// TIA Portal V15.1 export
// export: Created 2024-06-21T08:41:24.854849Z, ExportSetting WithDefaults, DisplayName Totally Integrated Automation Portal, DisplayVersion V15.1 Update 5, DisplayName TIA Portal Openness, DisplayVersion V15.1 Update 5, DisplayName SINAMICS Startdrive Advanced, DisplayVersion V15.1, DisplayName G130, G150, S120, S150, SINAMICS MV, S210, DisplayVersion V15.1, DisplayName G110M, G120, G120C, G120D, G120P, DisplayVersion V15.1, DisplayName STEP 7 Professional, DisplayVersion V15.1 Update 5, DisplayName STEP 7 Safety, DisplayVersion V15.1, DisplayName WinCC Professional, DisplayVersion V15.1 Update 5, DisplayName SIMATIC Visualization Architect, DisplayVersion V15.1
FUNCTION "209230ZM01" : Void   // FC400, FBD
TITLE = 209230ZM01 ModeZone
{ S7_Optimized_Access := 'FALSE' }
AUTHOR : VCG
NAME : Mot001
VERSION : 0.1
// stored: AutoNumber false, IsIECCheckEnabled false, SetENOAutomatically False, UDAEnableTagReadback false
   VAR_OUTPUT
      O_AlarmA : Bool;   // Alarm A
      O_AlarmB : Bool;   // Alarm B
      O_AlarmC : Bool;   // Alarm C
      O_AlarmD : Bool;   // Alarm D
      O_AlarmABCondition : Bool;   // Alarms resetable
      H_IAnim : Word;   // Animation bits to Icon in WinCC
   END_VAR
   VAR_TEMP   // added for the SCL form of the ladder/FBD networks
      _w1 : Bool;
      _w2 : Bool;
   END_VAR
BEGIN

REGION Network 1: **** 1 - Inputs **** HMI Commands
   // HMI Commands from the WinCC
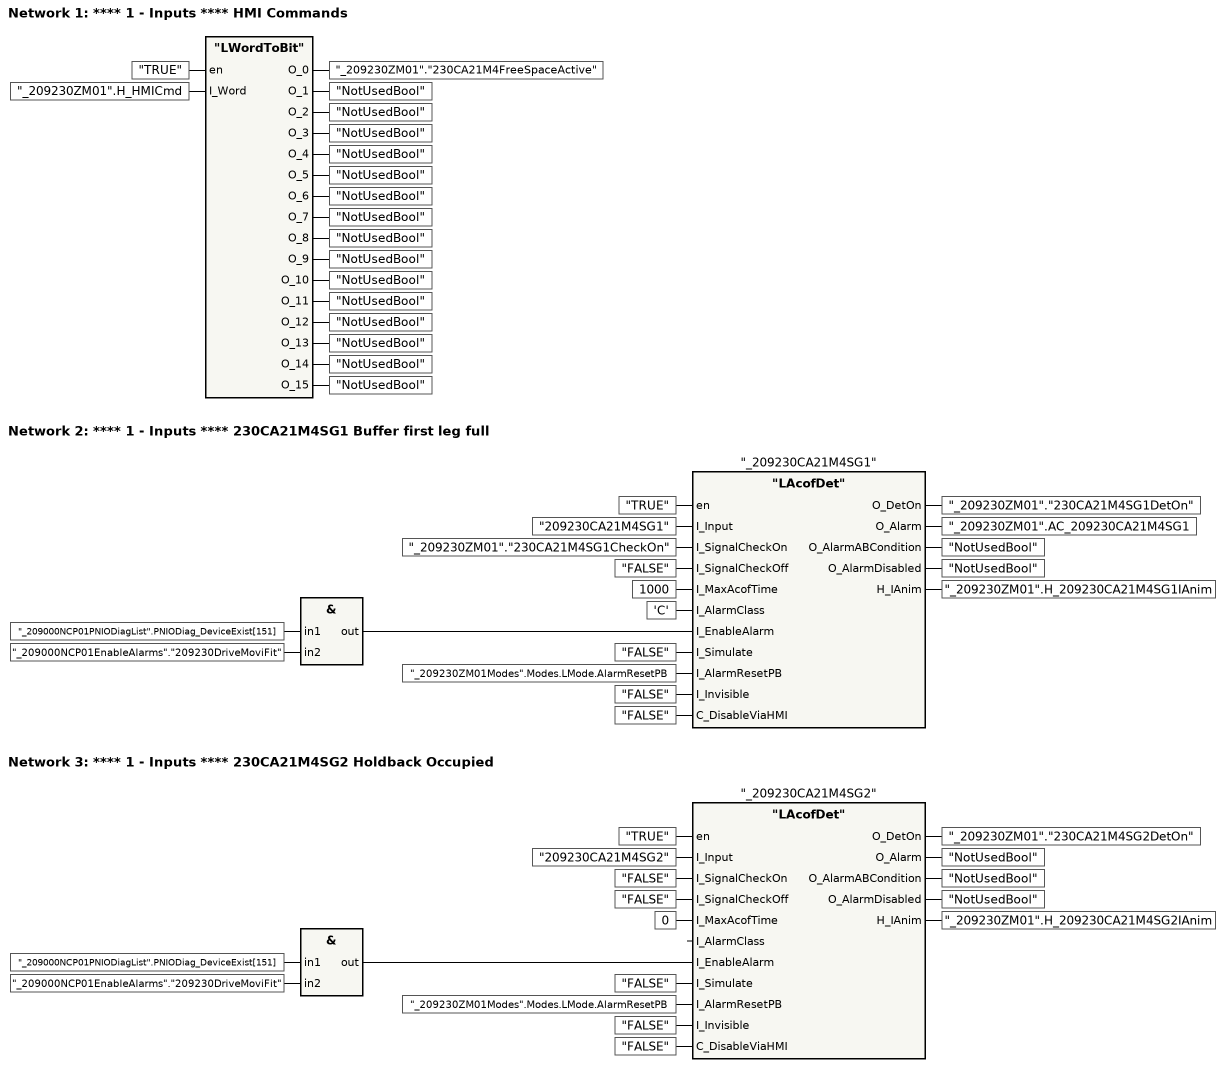
   IF "TRUE" THEN
       "LWordToBit"(I_Word := "_209230ZM01".H_HMICmd,
                    O_0 => "_209230ZM01"."230CA21M4FreeSpaceActive",
                    O_1 => "NotUsedBool",
                    O_2 => "NotUsedBool",
                    O_3 => "NotUsedBool",
                    O_4 => "NotUsedBool",
                    O_5 => "NotUsedBool",
                    O_6 => "NotUsedBool",
                    O_7 => "NotUsedBool",
                    O_8 => "NotUsedBool",
                    O_9 => "NotUsedBool",
                    O_10 => "NotUsedBool",
                    O_11 => "NotUsedBool",
                    O_12 => "NotUsedBool",
                    O_13 => "NotUsedBool",
                    O_14 => "NotUsedBool",
                    O_15 => "NotUsedBool");
   END_IF;
END_REGION

REGION Network 2: **** 1 - Inputs **** 230CA21M4SG1 Buffer first leg full
   IF "TRUE" THEN
       "_209230CA21M4SG1"(I_Input := "209230CA21M4SG1",   // "LAcofDet"
                          I_SignalCheckOn := "_209230ZM01"."230CA21M4SG1CheckOn",
                          I_SignalCheckOff := "FALSE",
                          I_MaxAcofTime := 1000,
                          I_AlarmClass := 'C',
                          I_EnableAlarm := "_209000NCP01PNIODiagList".PNIODiag_DeviceExist[151] AND "_209000NCP01EnableAlarms"."209230DriveMoviFit",
                          I_Simulate := "FALSE",
                          I_AlarmResetPB := "_209230ZM01Modes".Modes.LMode.AlarmResetPB,
                          I_Invisible := "FALSE",
                          C_DisableViaHMI := "FALSE",
                          O_DetOn => "_209230ZM01"."230CA21M4SG1DetOn",
                          O_Alarm => "_209230ZM01".AC_209230CA21M4SG1,
                          O_AlarmABCondition => "NotUsedBool",
                          O_AlarmDisabled => "NotUsedBool",
                          H_IAnim => "_209230ZM01".H_209230CA21M4SG1IAnim);
   END_IF;
END_REGION

REGION Network 3: **** 1 - Inputs **** 230CA21M4SG2 Holdback Occupied
   IF "TRUE" THEN
       "_209230CA21M4SG2"(I_Input := "209230CA21M4SG2",   // "LAcofDet"
                          I_SignalCheckOn := "FALSE",
                          I_SignalCheckOff := "FALSE",
                          I_MaxAcofTime := 0,
                          I_EnableAlarm := "_209000NCP01PNIODiagList".PNIODiag_DeviceExist[151] AND "_209000NCP01EnableAlarms"."209230DriveMoviFit",
                          I_Simulate := "FALSE",
                          I_AlarmResetPB := "_209230ZM01Modes".Modes.LMode.AlarmResetPB,
                          I_Invisible := "FALSE",
                          C_DisableViaHMI := "FALSE",
                          O_DetOn => "_209230ZM01"."230CA21M4SG2DetOn",
                          O_Alarm => "NotUsedBool",
                          O_AlarmABCondition => "NotUsedBool",
                          O_AlarmDisabled => "NotUsedBool",
                          H_IAnim => "_209230ZM01".H_209230CA21M4SG2IAnim);
   END_IF;
END_REGION

REGION Network 4: **** 1 - Inputs **** 230CA21M4SG3 OK to close Holdback
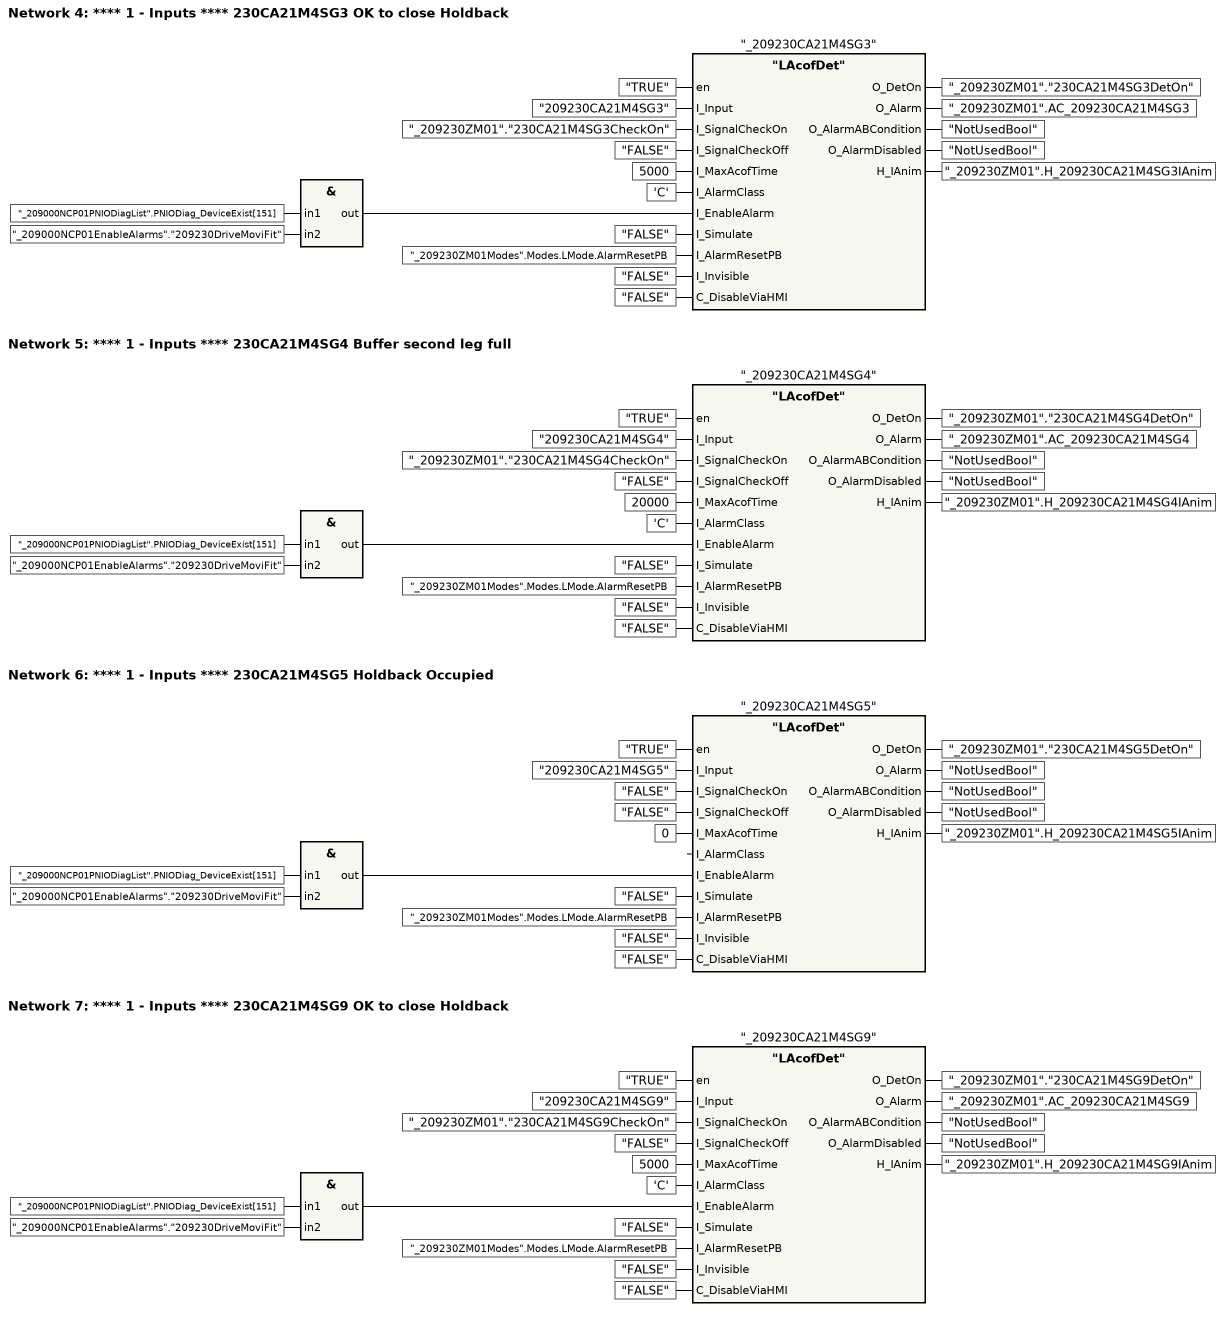
   IF "TRUE" THEN
       "_209230CA21M4SG3"(I_Input := "209230CA21M4SG3",   // "LAcofDet"
                          I_SignalCheckOn := "_209230ZM01"."230CA21M4SG3CheckOn",
                          I_SignalCheckOff := "FALSE",
                          I_MaxAcofTime := 5000,
                          I_AlarmClass := 'C',
                          I_EnableAlarm := "_209000NCP01PNIODiagList".PNIODiag_DeviceExist[151] AND "_209000NCP01EnableAlarms"."209230DriveMoviFit",
                          I_Simulate := "FALSE",
                          I_AlarmResetPB := "_209230ZM01Modes".Modes.LMode.AlarmResetPB,
                          I_Invisible := "FALSE",
                          C_DisableViaHMI := "FALSE",
                          O_DetOn => "_209230ZM01"."230CA21M4SG3DetOn",
                          O_Alarm => "_209230ZM01".AC_209230CA21M4SG3,
                          O_AlarmABCondition => "NotUsedBool",
                          O_AlarmDisabled => "NotUsedBool",
                          H_IAnim => "_209230ZM01".H_209230CA21M4SG3IAnim);
   END_IF;
END_REGION

REGION Network 5: **** 1 - Inputs **** 230CA21M4SG4 Buffer second leg full
   IF "TRUE" THEN
       "_209230CA21M4SG4"(I_Input := "209230CA21M4SG4",   // "LAcofDet"
                          I_SignalCheckOn := "_209230ZM01"."230CA21M4SG4CheckOn",
                          I_SignalCheckOff := "FALSE",
                          I_MaxAcofTime := 20000,
                          I_AlarmClass := 'C',
                          I_EnableAlarm := "_209000NCP01PNIODiagList".PNIODiag_DeviceExist[151] AND "_209000NCP01EnableAlarms"."209230DriveMoviFit",
                          I_Simulate := "FALSE",
                          I_AlarmResetPB := "_209230ZM01Modes".Modes.LMode.AlarmResetPB,
                          I_Invisible := "FALSE",
                          C_DisableViaHMI := "FALSE",
                          O_DetOn => "_209230ZM01"."230CA21M4SG4DetOn",
                          O_Alarm => "_209230ZM01".AC_209230CA21M4SG4,
                          O_AlarmABCondition => "NotUsedBool",
                          O_AlarmDisabled => "NotUsedBool",
                          H_IAnim => "_209230ZM01".H_209230CA21M4SG4IAnim);
   END_IF;
END_REGION

REGION Network 6: **** 1 - Inputs **** 230CA21M4SG5 Holdback Occupied
   IF "TRUE" THEN
       "_209230CA21M4SG5"(I_Input := "209230CA21M4SG5",   // "LAcofDet"
                          I_SignalCheckOn := "FALSE",
                          I_SignalCheckOff := "FALSE",
                          I_MaxAcofTime := 0,
                          I_EnableAlarm := "_209000NCP01PNIODiagList".PNIODiag_DeviceExist[151] AND "_209000NCP01EnableAlarms"."209230DriveMoviFit",
                          I_Simulate := "FALSE",
                          I_AlarmResetPB := "_209230ZM01Modes".Modes.LMode.AlarmResetPB,
                          I_Invisible := "FALSE",
                          C_DisableViaHMI := "FALSE",
                          O_DetOn => "_209230ZM01"."230CA21M4SG5DetOn",
                          O_Alarm => "NotUsedBool",
                          O_AlarmABCondition => "NotUsedBool",
                          O_AlarmDisabled => "NotUsedBool",
                          H_IAnim => "_209230ZM01".H_209230CA21M4SG5IAnim);
   END_IF;
END_REGION

REGION Network 7: **** 1 - Inputs **** 230CA21M4SG9 OK to close Holdback
   IF "TRUE" THEN
       "_209230CA21M4SG9"(I_Input := "209230CA21M4SG9",   // "LAcofDet"
                          I_SignalCheckOn := "_209230ZM01"."230CA21M4SG9CheckOn",
                          I_SignalCheckOff := "FALSE",
                          I_MaxAcofTime := 5000,
                          I_AlarmClass := 'C',
                          I_EnableAlarm := "_209000NCP01PNIODiagList".PNIODiag_DeviceExist[151] AND "_209000NCP01EnableAlarms"."209230DriveMoviFit",
                          I_Simulate := "FALSE",
                          I_AlarmResetPB := "_209230ZM01Modes".Modes.LMode.AlarmResetPB,
                          I_Invisible := "FALSE",
                          C_DisableViaHMI := "FALSE",
                          O_DetOn => "_209230ZM01"."230CA21M4SG9DetOn",
                          O_Alarm => "_209230ZM01".AC_209230CA21M4SG9,
                          O_AlarmABCondition => "NotUsedBool",
                          O_AlarmDisabled => "NotUsedBool",
                          H_IAnim => "_209230ZM01".H_209230CA21M4SG9IAnim);
   END_IF;
END_REGION

REGION Network 8: **** 1 - Inputs **** 230CA21M4 Buffer Full
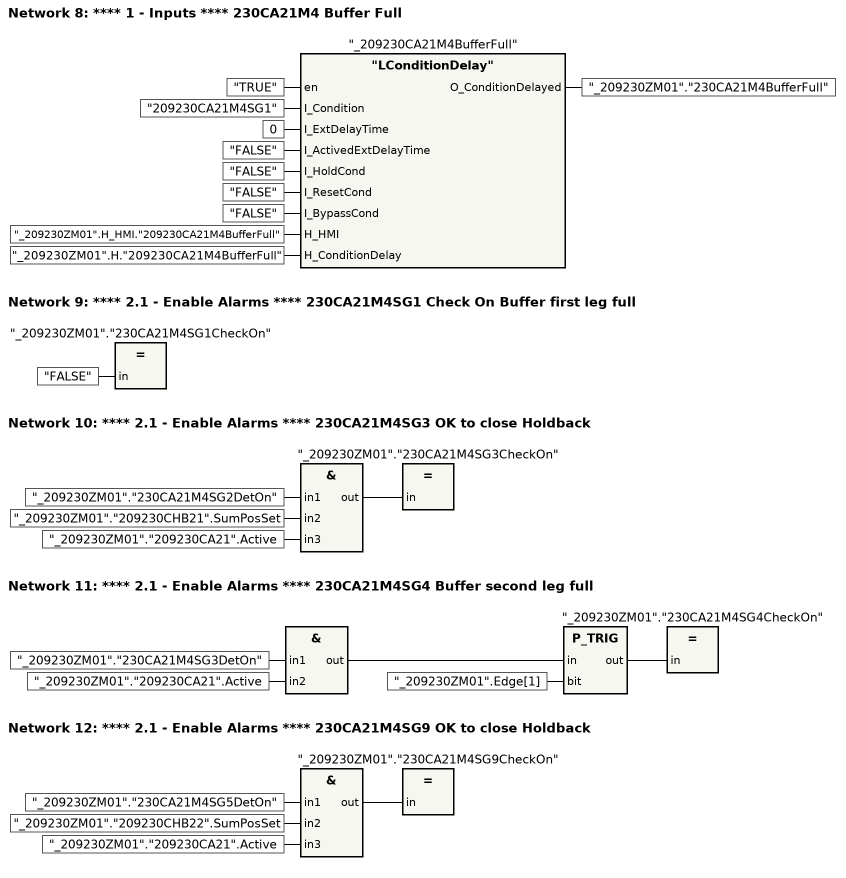
   IF "TRUE" THEN
       "_209230CA21M4BufferFull"(I_Condition := "209230CA21M4SG1",   // "LConditionDelay"
                               I_ExtDelayTime := 0,
                               I_ActivedExtDelayTime := "FALSE",
                               I_HoldCond := "FALSE",
                               I_ResetCond := "FALSE",
                               I_BypassCond := "FALSE",
                               H_HMI := "_209230ZM01".H_HMI."209230CA21M4BufferFull",
                               H_ConditionDelay := "_209230ZM01".H."209230CA21M4BufferFull",
                               O_ConditionDelayed => "_209230ZM01"."230CA21M4BufferFull");
   END_IF;
END_REGION

REGION Network 9: **** 2.1 - Enable Alarms **** 230CA21M4SG1 Check On Buffer first leg full
   "_209230ZM01"."230CA21M4SG1CheckOn" := "FALSE";
END_REGION

REGION Network 10: **** 2.1 - Enable Alarms **** 230CA21M4SG3 OK to close Holdback
   "_209230ZM01"."230CA21M4SG3CheckOn" := "_209230ZM01"."230CA21M4SG2DetOn" AND "_209230ZM01"."209230CHB21".SumPosSet AND "_209230ZM01"."209230CA21".Active;
END_REGION

REGION Network 11: **** 2.1 - Enable Alarms **** 230CA21M4SG4 Buffer second leg full
   #_w1 := "_209230ZM01"."230CA21M4SG3DetOn" AND "_209230ZM01"."209230CA21".Active;
   #_w2 := #_w1 AND NOT "_209230ZM01".Edge[1];   // rising edge
   "_209230ZM01".Edge[1] := #_w1;
   "_209230ZM01"."230CA21M4SG4CheckOn" := #_w2;
END_REGION

REGION Network 12: **** 2.1 - Enable Alarms **** 230CA21M4SG9 OK to close Holdback
   "_209230ZM01"."230CA21M4SG9CheckOn" := "_209230ZM01"."230CA21M4SG5DetOn" AND "_209230ZM01"."209230CHB22".SumPosSet AND "_209230ZM01"."209230CA21".Active;
END_REGION

REGION Network 13: **** 3.1 - Communication - Other Systems **** Supervision
   // Supervision
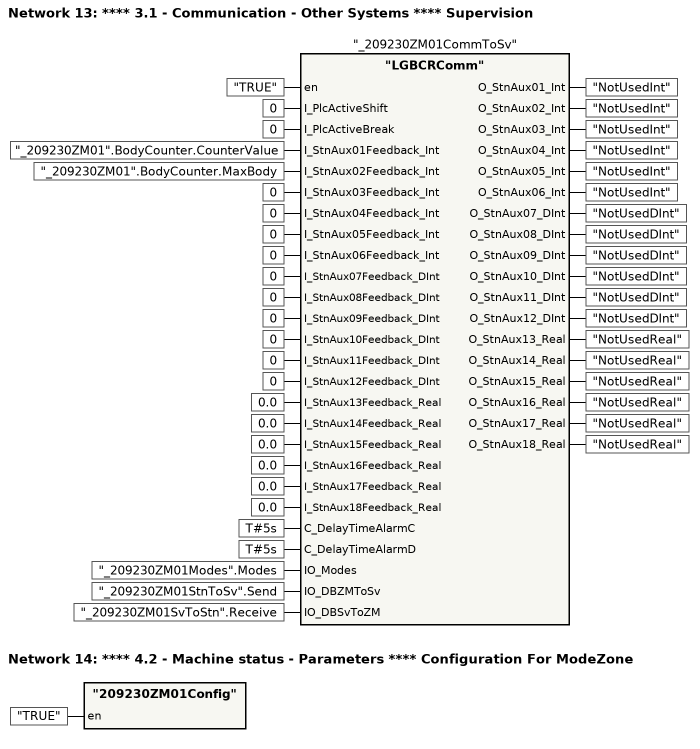
   IF "TRUE" THEN
       "_209230ZM01CommToSv"(I_PlcActiveShift := 0,   // "LGBCRComm"
                             I_PlcActiveBreak := 0,
                             I_StnAux01Feedback_Int := "_209230ZM01".BodyCounter.CounterValue,
                             I_StnAux02Feedback_Int := "_209230ZM01".BodyCounter.MaxBody,
                             I_StnAux03Feedback_Int := 0,
                             I_StnAux04Feedback_Int := 0,
                             I_StnAux05Feedback_Int := 0,
                             I_StnAux06Feedback_Int := 0,
                             I_StnAux07Feedback_DInt := 0,
                             I_StnAux08Feedback_DInt := 0,
                             I_StnAux09Feedback_DInt := 0,
                             I_StnAux10Feedback_DInt := 0,
                             I_StnAux11Feedback_DInt := 0,
                             I_StnAux12Feedback_DInt := 0,
                             I_StnAux13Feedback_Real := 0.0,
                             I_StnAux14Feedback_Real := 0.0,
                             I_StnAux15Feedback_Real := 0.0,
                             I_StnAux16Feedback_Real := 0.0,
                             I_StnAux17Feedback_Real := 0.0,
                             I_StnAux18Feedback_Real := 0.0,
                             C_DelayTimeAlarmC := T#5s,
                             C_DelayTimeAlarmD := T#5s,
                             IO_Modes := "_209230ZM01Modes".Modes,
                             IO_DBZMToSv := "_209230ZM01StnToSv".Send,
                             IO_DBSvToZM := "_209230ZM01SvToStn".Receive,
                             O_StnAux01_Int => "NotUsedInt",
                             O_StnAux02_Int => "NotUsedInt",
                             O_StnAux03_Int => "NotUsedInt",
                             O_StnAux04_Int => "NotUsedInt",
                             O_StnAux05_Int => "NotUsedInt",
                             O_StnAux06_Int => "NotUsedInt",
                             O_StnAux07_DInt => "NotUsedDInt",
                             O_StnAux08_DInt => "NotUsedDInt",
                             O_StnAux09_DInt => "NotUsedDInt",
                             O_StnAux10_DInt => "NotUsedDInt",
                             O_StnAux11_DInt => "NotUsedDInt",
                             O_StnAux12_DInt => "NotUsedDInt",
                             O_StnAux13_Real => "NotUsedReal",
                             O_StnAux14_Real => "NotUsedReal",
                             O_StnAux15_Real => "NotUsedReal",
                             O_StnAux16_Real => "NotUsedReal",
                             O_StnAux17_Real => "NotUsedReal",
                             O_StnAux18_Real => "NotUsedReal");
   END_IF;
END_REGION

REGION Network 14: **** 4.2 - Machine status - Parameters **** Configuration For ModeZone
   // Configuration of equipment for ModeZone
   IF "TRUE" THEN "209230ZM01Config"(); END_IF;
END_REGION

REGION Network 15: **** 4.2 - Machine status - Parameters **** Body Counter
   // Body Counter
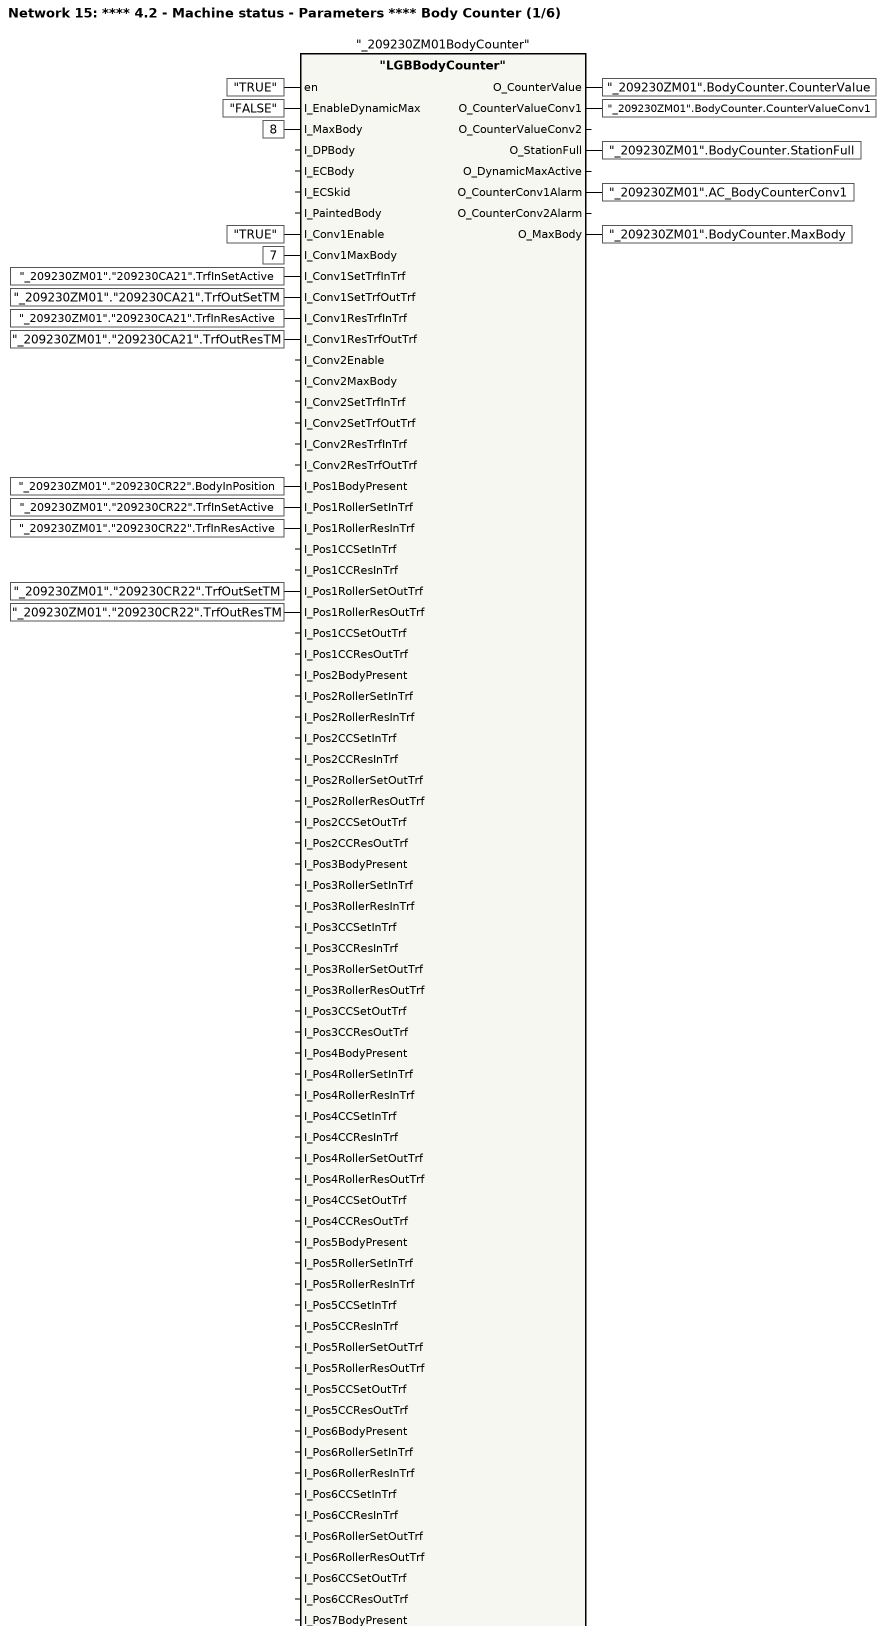
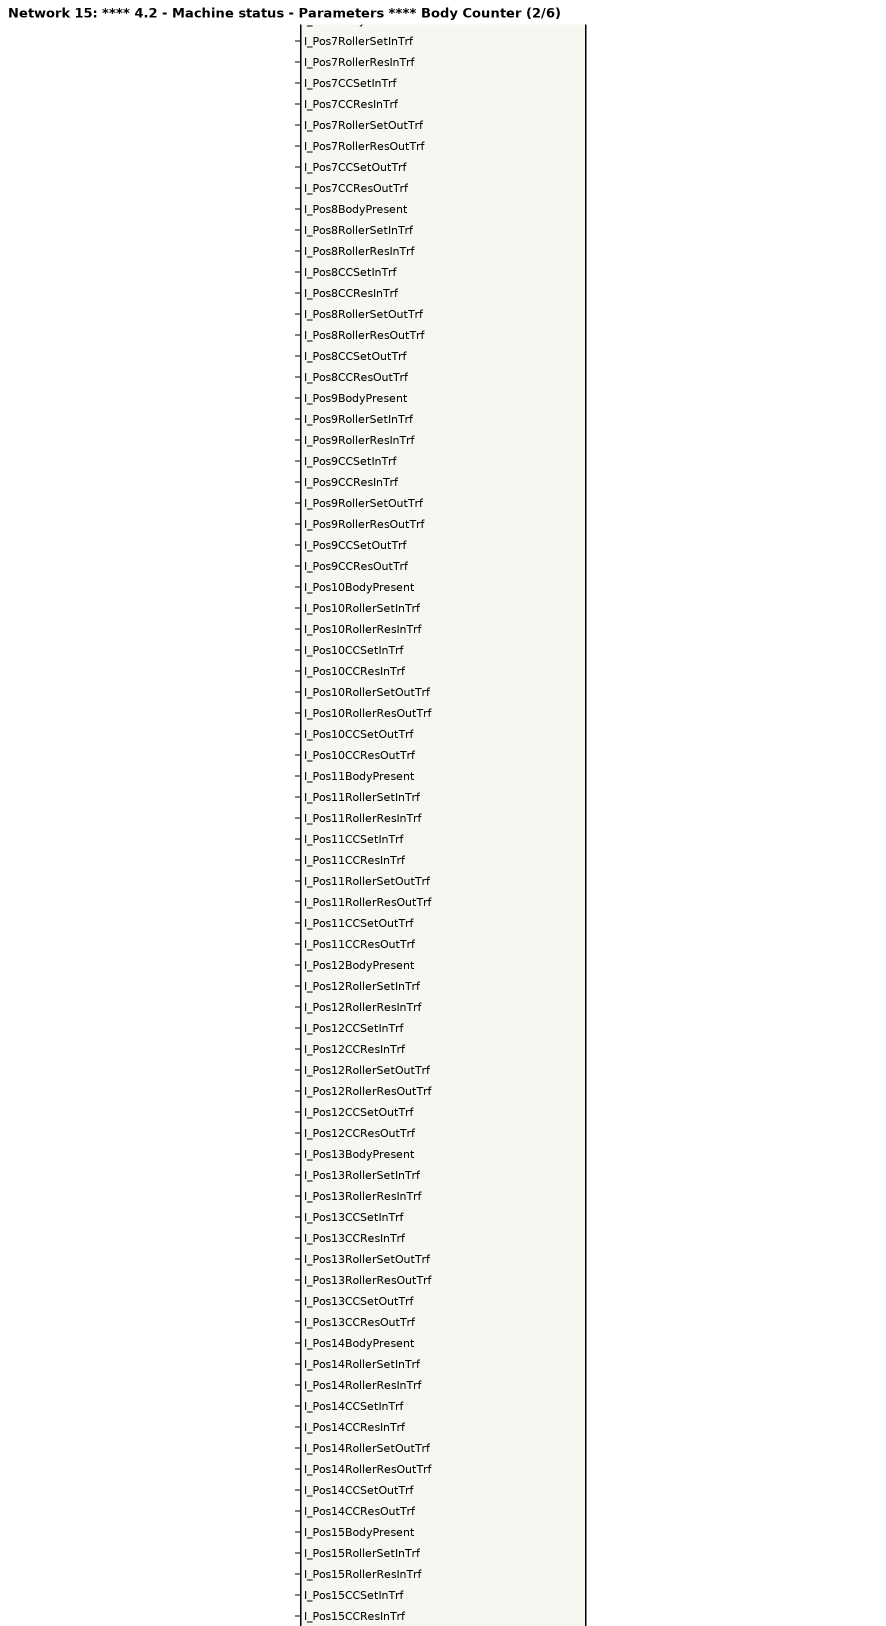
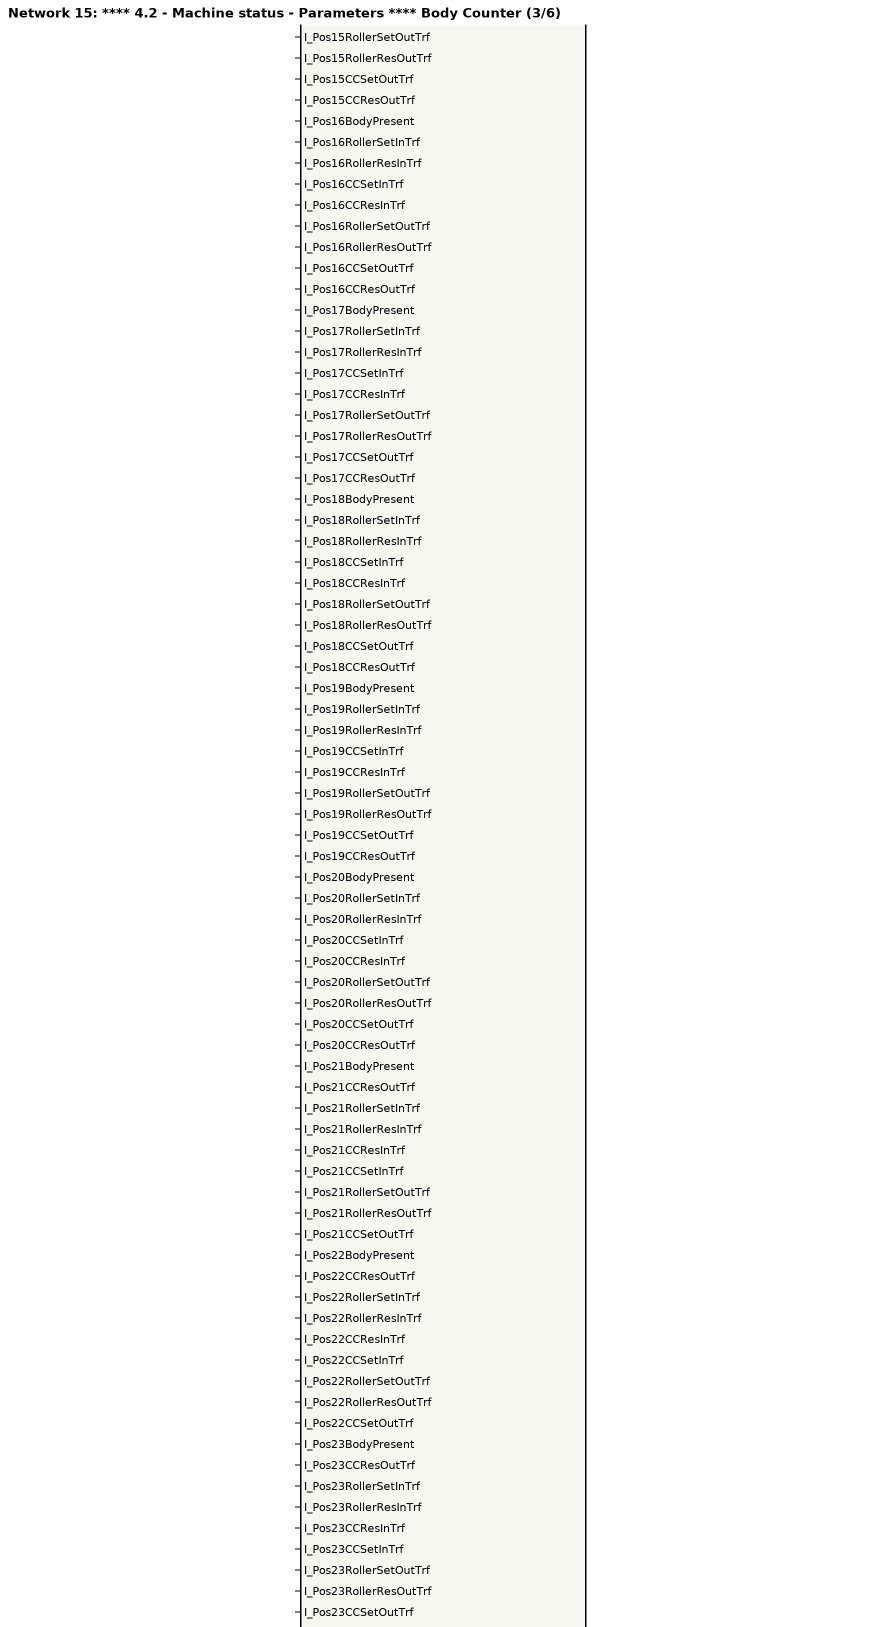
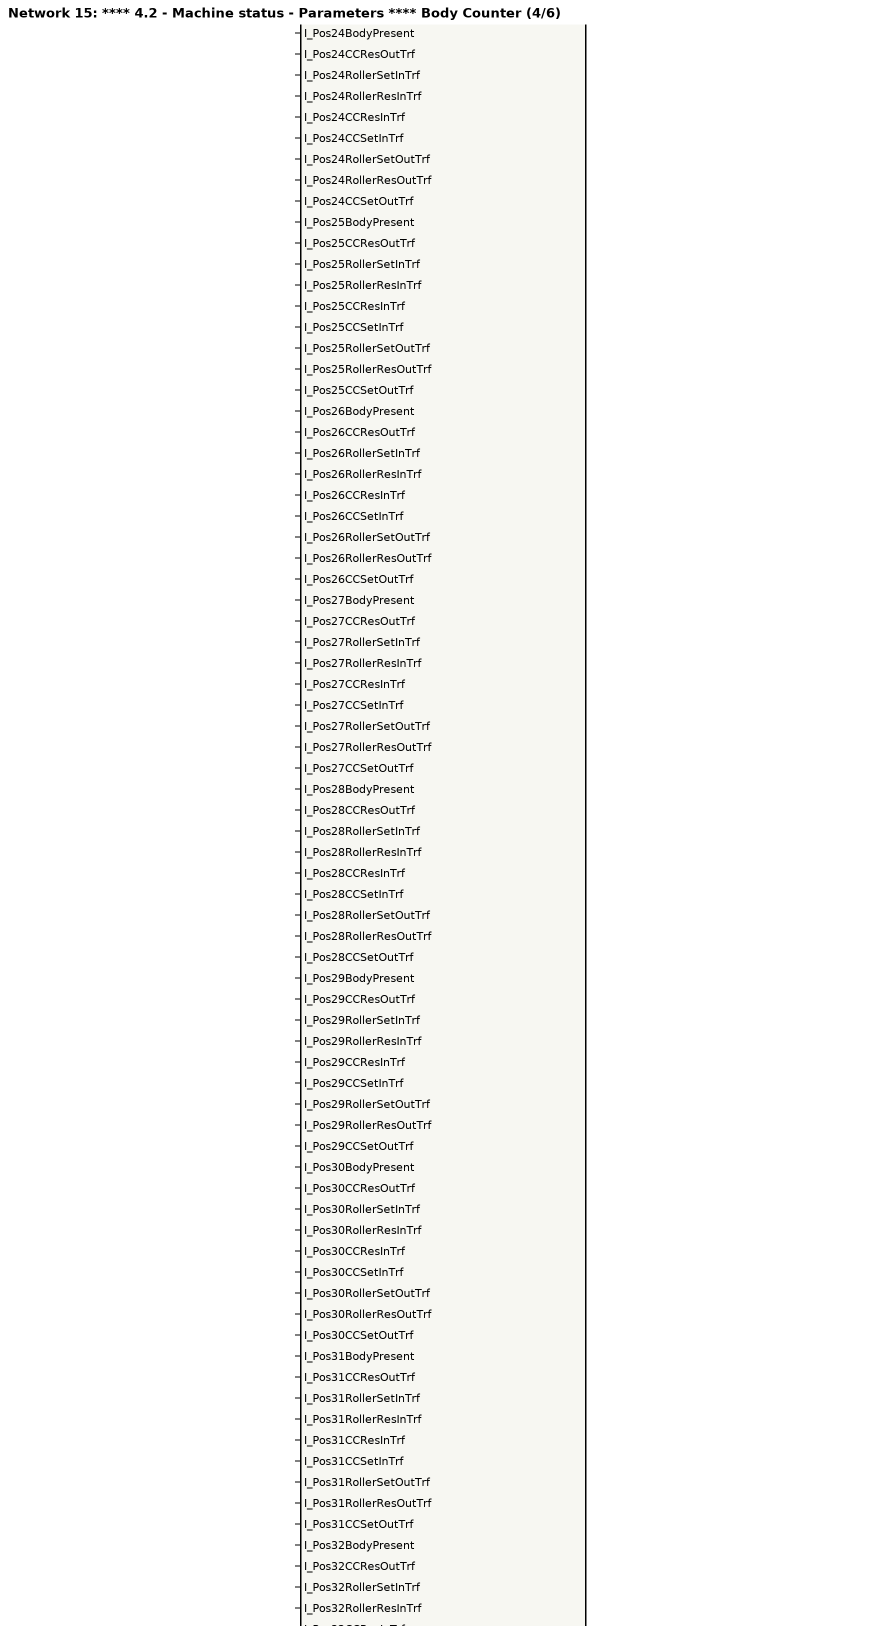
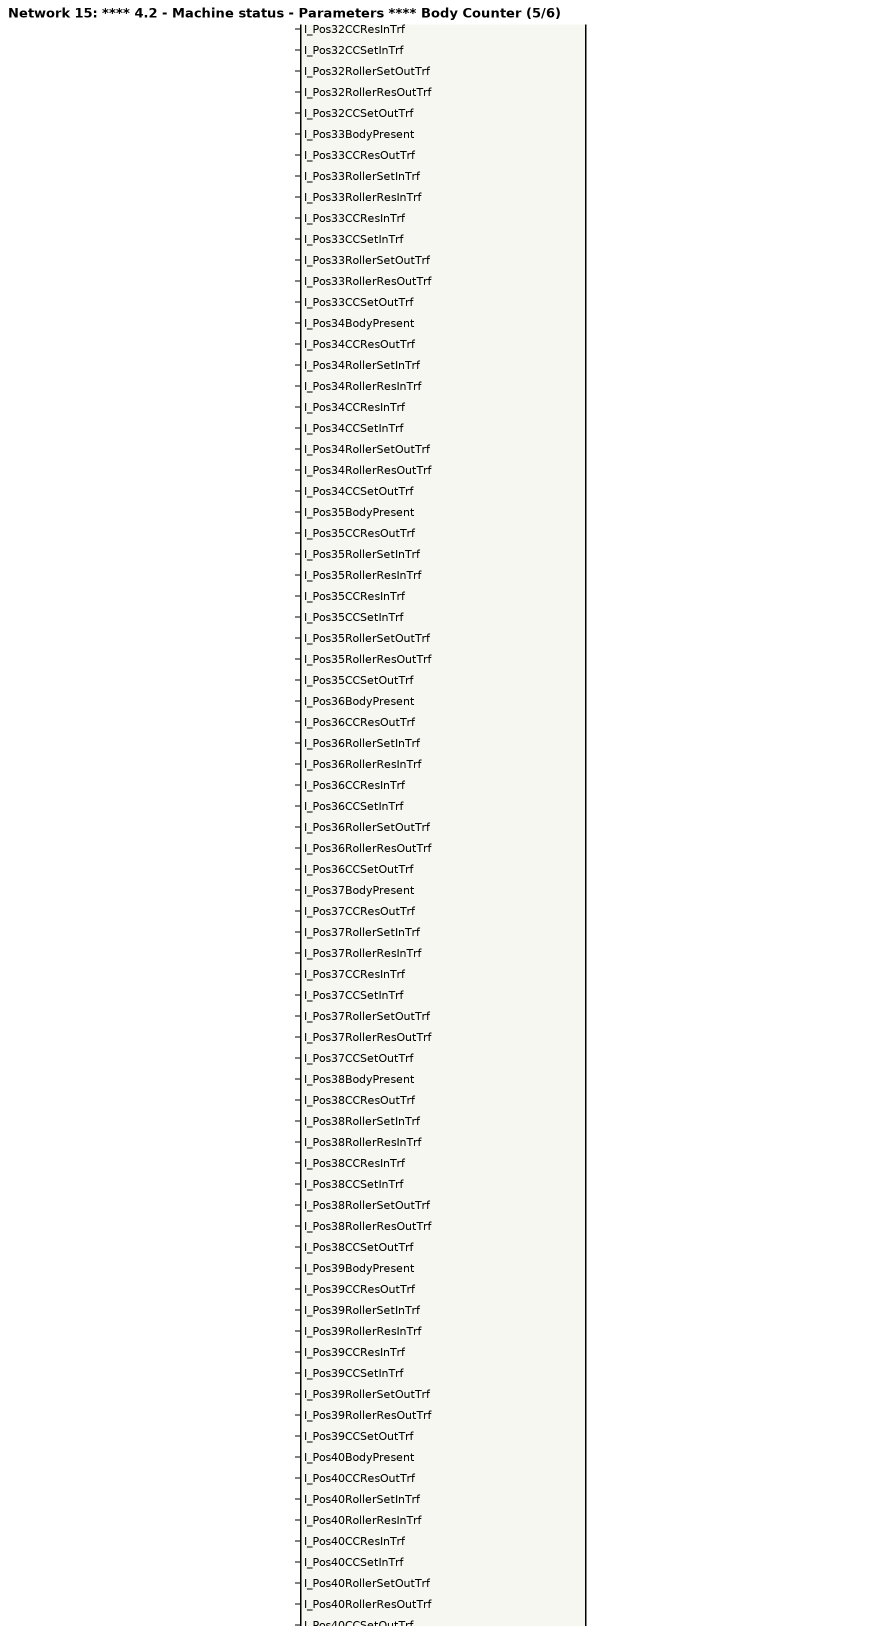
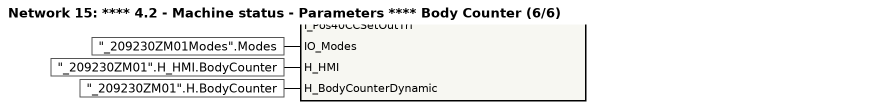
   IF "TRUE" THEN
       "_209230ZM01BodyCounter"(I_EnableDynamicMax := "FALSE",   // "LGBBodyCounter"
                               I_MaxBody := 8,
                               I_Conv1Enable := "TRUE",
                               I_Conv1MaxBody := 7,
                               I_Conv1SetTrfInTrf := "_209230ZM01"."209230CA21".TrfInSetActive,
                               I_Conv1SetTrfOutTrf := "_209230ZM01"."209230CA21".TrfOutSetTM,
                               I_Conv1ResTrfInTrf := "_209230ZM01"."209230CA21".TrfInResActive,
                               I_Conv1ResTrfOutTrf := "_209230ZM01"."209230CA21".TrfOutResTM,
                               I_Pos1BodyPresent := "_209230ZM01"."209230CR22".BodyInPosition,
                               I_Pos1RollerSetInTrf := "_209230ZM01"."209230CR22".TrfInSetActive,
                               I_Pos1RollerResInTrf := "_209230ZM01"."209230CR22".TrfInResActive,
                               I_Pos1RollerSetOutTrf := "_209230ZM01"."209230CR22".TrfOutSetTM,
                               I_Pos1RollerResOutTrf := "_209230ZM01"."209230CR22".TrfOutResTM,
                               IO_Modes := "_209230ZM01Modes".Modes,
                               H_HMI := "_209230ZM01".H_HMI.BodyCounter,
                               H_BodyCounterDynamic := "_209230ZM01".H.BodyCounter,
                               O_CounterValue => "_209230ZM01".BodyCounter.CounterValue,
                               O_CounterValueConv1 => "_209230ZM01".BodyCounter.CounterValueConv1,
                               O_StationFull => "_209230ZM01".BodyCounter.StationFull,
                               O_CounterConv1Alarm => "_209230ZM01".AC_BodyCounterConv1,
                               O_MaxBody => "_209230ZM01".BodyCounter.MaxBody);
   END_IF;
END_REGION

REGION Network 16: **** 4.4 - Machine Status - Calculation **** Home Position Station
   // Home position of the ModeZone
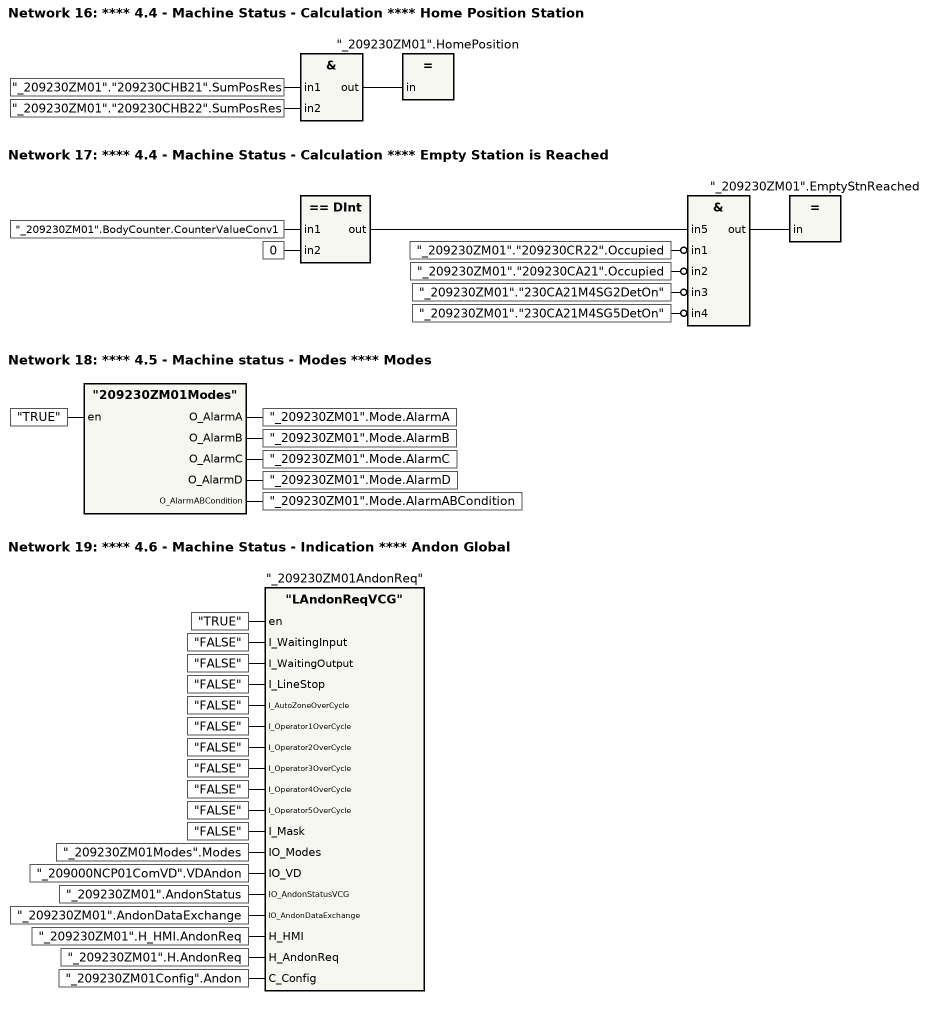
   "_209230ZM01".HomePosition := "_209230ZM01"."209230CHB21".SumPosRes AND "_209230ZM01"."209230CHB22".SumPosRes;
END_REGION

REGION Network 17: **** 4.4 - Machine Status - Calculation **** Empty Station is Reached
   // Empty Station
   "_209230ZM01".EmptyStnReached := ("_209230ZM01".BodyCounter.CounterValueConv1 = 0) AND NOT "_209230ZM01"."209230CR22".Occupied AND NOT "_209230ZM01"."209230CA21".Occupied AND NOT "_209230ZM01"."230CA21M4SG2DetOn" AND NOT "_209230ZM01"."230CA21M4SG5DetOn";
END_REGION

REGION Network 18: **** 4.5 - Machine status - Modes **** Modes
   // Modes
   IF "TRUE" THEN
       "209230ZM01Modes"(O_AlarmA => "_209230ZM01".Mode.AlarmA,
                         O_AlarmB => "_209230ZM01".Mode.AlarmB,
                         O_AlarmC => "_209230ZM01".Mode.AlarmC,
                         O_AlarmD => "_209230ZM01".Mode.AlarmD,
                         O_AlarmABCondition => "_209230ZM01".Mode.AlarmABCondition);
   END_IF;
END_REGION

REGION Network 19: **** 4.6 - Machine Status - Indication **** Andon Global
   // Request Andon Call
   IF "TRUE" THEN
       "_209230ZM01AndonReq"(I_WaitingInput := "FALSE",   // "LAndonReqVCG"
                             I_WaitingOutput := "FALSE",
                             I_LineStop := "FALSE",
                             I_AutoZoneOverCycle := "FALSE",
                             I_Operator1OverCycle := "FALSE",
                             I_Operator2OverCycle := "FALSE",
                             I_Operator3OverCycle := "FALSE",
                             I_Operator4OverCycle := "FALSE",
                             I_Operator5OverCycle := "FALSE",
                             I_Mask := "FALSE",
                             IO_Modes := "_209230ZM01Modes".Modes,
                             IO_VD := "_209000NCP01ComVD".VDAndon,
                             IO_AndonStatusVCG := "_209230ZM01".AndonStatus,
                             IO_AndonDataExchange := "_209230ZM01".AndonDataExchange,
                             H_HMI := "_209230ZM01".H_HMI.AndonReq,
                             H_AndonReq := "_209230ZM01".H.AndonReq,
                             C_Config := "_209230ZM01Config".Andon);
   END_IF;
END_REGION

REGION Network 20: **** 4.6 - Machine status - Indications **** Icon animation
   // Icon animation
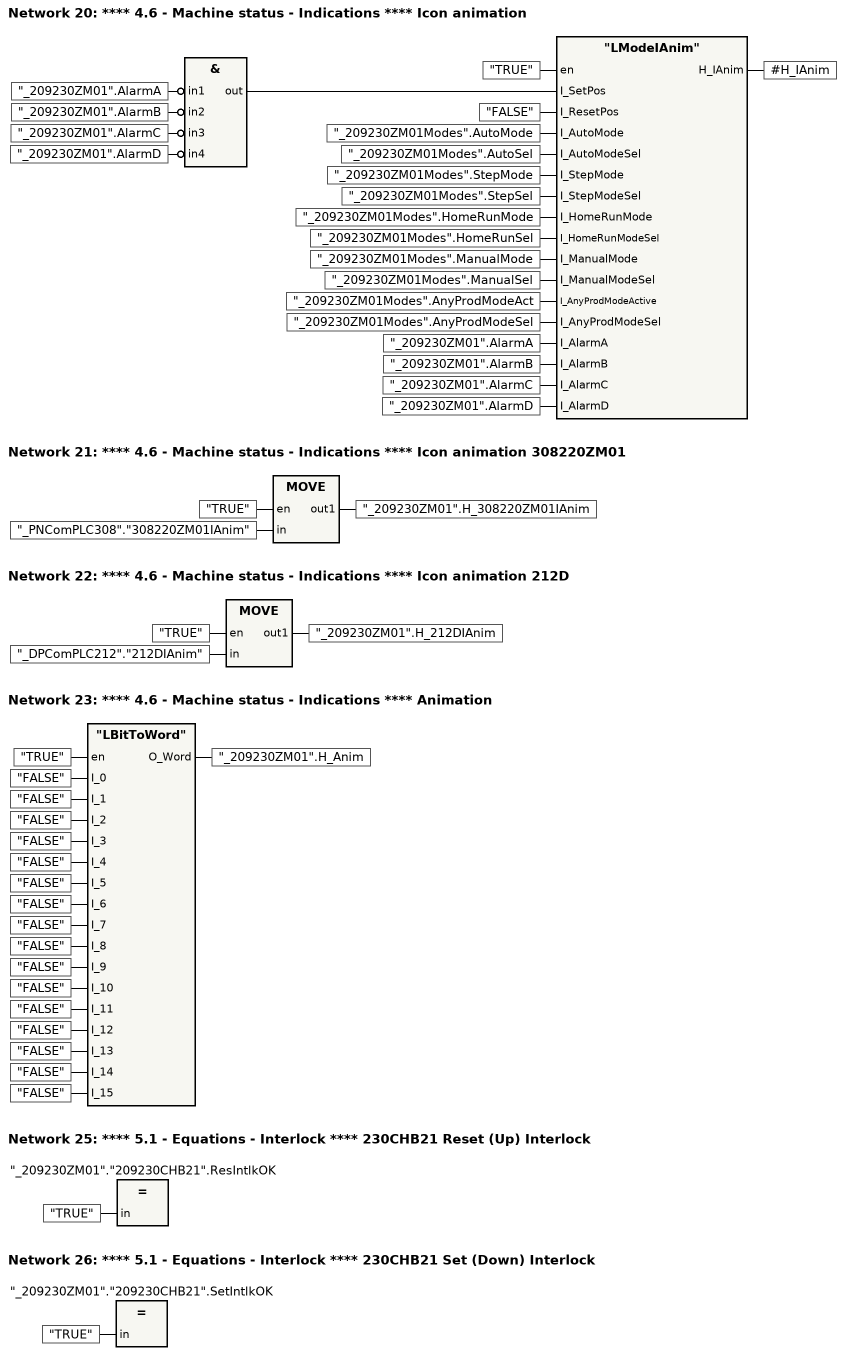
   IF "TRUE" THEN
       "LModeIAnim"(I_SetPos := NOT "_209230ZM01".AlarmA AND NOT "_209230ZM01".AlarmB AND NOT "_209230ZM01".AlarmC AND NOT "_209230ZM01".AlarmD,
                    I_ResetPos := "FALSE",
                    I_AutoMode := "_209230ZM01Modes".AutoMode,
                    I_AutoModeSel := "_209230ZM01Modes".AutoSel,
                    I_StepMode := "_209230ZM01Modes".StepMode,
                    I_StepModeSel := "_209230ZM01Modes".StepSel,
                    I_HomeRunMode := "_209230ZM01Modes".HomeRunMode,
                    I_HomeRunModeSel := "_209230ZM01Modes".HomeRunSel,
                    I_ManualMode := "_209230ZM01Modes".ManualMode,
                    I_ManualModeSel := "_209230ZM01Modes".ManualSel,
                    I_AnyProdModeActive := "_209230ZM01Modes".AnyProdModeAct,
                    I_AnyProdModeSel := "_209230ZM01Modes".AnyProdModeSel,
                    I_AlarmA := "_209230ZM01".AlarmA,
                    I_AlarmB := "_209230ZM01".AlarmB,
                    I_AlarmC := "_209230ZM01".AlarmC,
                    I_AlarmD := "_209230ZM01".AlarmD,
                    H_IAnim => #H_IAnim);
   END_IF;
END_REGION

REGION Network 21: **** 4.6 - Machine status - Indications **** Icon animation 308220ZM01
   // Icon animation
   IF "TRUE" THEN "_209230ZM01".H_308220ZM01IAnim := "_PNComPLC308"."308220ZM01IAnim"; END_IF;
END_REGION

REGION Network 22: **** 4.6 - Machine status - Indications **** Icon animation 212D
   // Icon animation
   IF "TRUE" THEN "_209230ZM01".H_212DIAnim := "_DPComPLC212"."212DIAnim"; END_IF;
END_REGION

REGION Network 23: **** 4.6 - Machine status - Indications **** Animation
   // Animation
   IF "TRUE" THEN
       "LBitToWord"(I_0 := "FALSE",
                    I_1 := "FALSE",
                    I_2 := "FALSE",
                    I_3 := "FALSE",
                    I_4 := "FALSE",
                    I_5 := "FALSE",
                    I_6 := "FALSE",
                    I_7 := "FALSE",
                    I_8 := "FALSE",
                    I_9 := "FALSE",
                    I_10 := "FALSE",
                    I_11 := "FALSE",
                    I_12 := "FALSE",
                    I_13 := "FALSE",
                    I_14 := "FALSE",
                    I_15 := "FALSE",
                    O_Word => "_209230ZM01".H_Anim);
   END_IF;
END_REGION

NETWORK
TITLE = **** 4.6 - Machine Status - Indications **** Animation DB number
// DB number
      OPN   "_209230ZM01";
      L     DBNO;
      T     "_209230ZM01".H_DBnr;

REGION Network 25: **** 5.1 - Equations - Interlock **** 230CHB21 Reset (Up) Interlock
   "_209230ZM01"."209230CHB21".ResIntlkOK := "TRUE";
END_REGION

REGION Network 26: **** 5.1 - Equations - Interlock **** 230CHB21 Set (Down) Interlock
   "_209230ZM01"."209230CHB21".SetIntlkOK := "TRUE";
END_REGION

REGION Network 27: **** 5.1 - Equations - Interlock **** 230CHB22 Reset (Up) Interlock
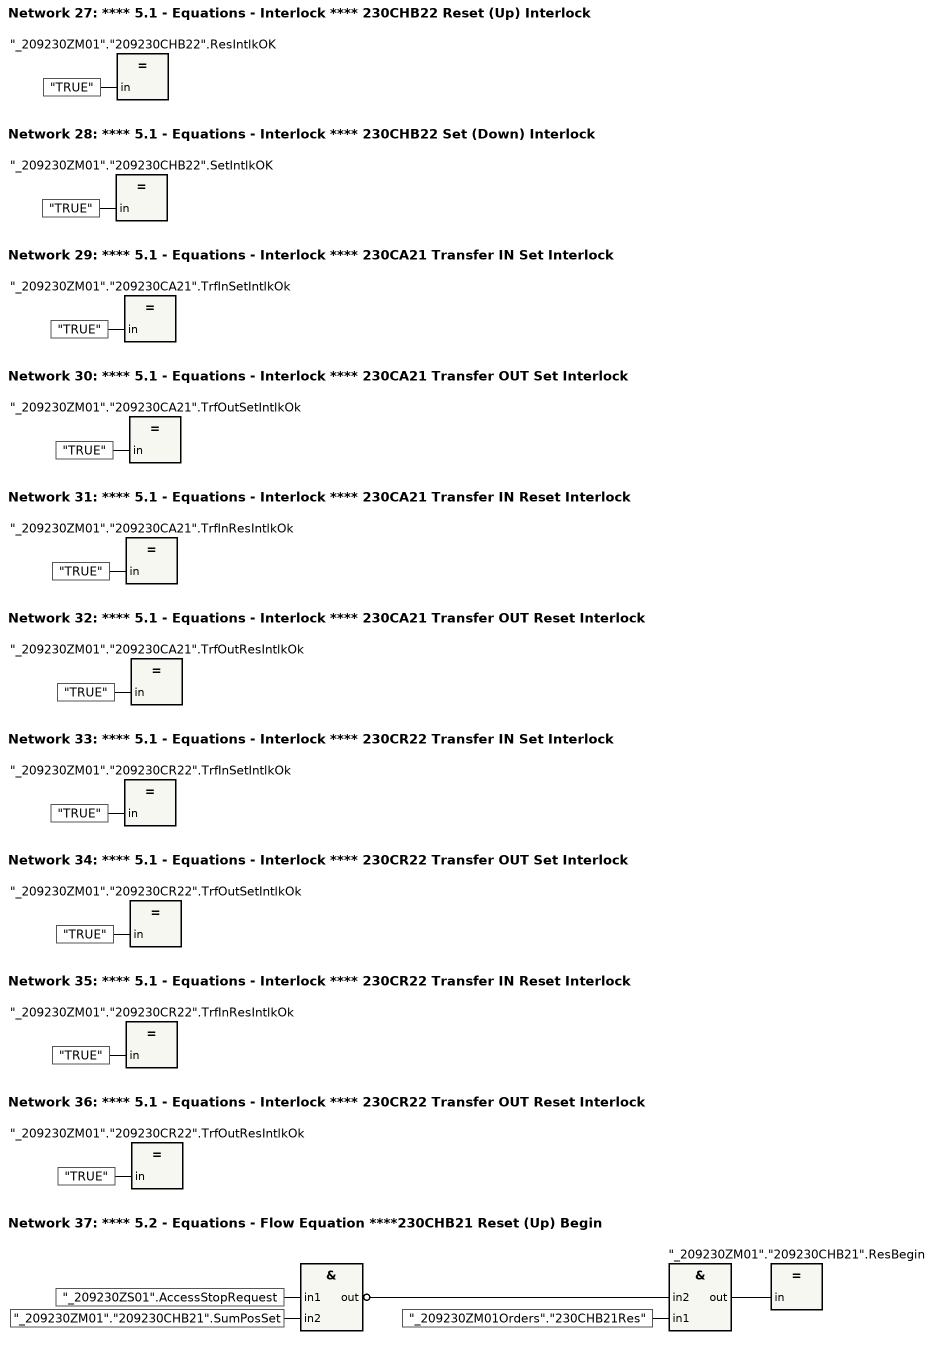
   "_209230ZM01"."209230CHB22".ResIntlkOK := "TRUE";
END_REGION

REGION Network 28: **** 5.1 - Equations - Interlock **** 230CHB22 Set (Down) Interlock
   "_209230ZM01"."209230CHB22".SetIntlkOK := "TRUE";
END_REGION

REGION Network 29: **** 5.1 - Equations - Interlock **** 230CA21 Transfer IN Set Interlock
   "_209230ZM01"."209230CA21".TrfInSetIntlkOk := "TRUE";
END_REGION

REGION Network 30: **** 5.1 - Equations - Interlock **** 230CA21 Transfer OUT Set Interlock
   "_209230ZM01"."209230CA21".TrfOutSetIntlkOk := "TRUE";
END_REGION

REGION Network 31: **** 5.1 - Equations - Interlock **** 230CA21 Transfer IN Reset Interlock
   "_209230ZM01"."209230CA21".TrfInResIntlkOk := "TRUE";
END_REGION

REGION Network 32: **** 5.1 - Equations - Interlock **** 230CA21 Transfer OUT Reset Interlock
   "_209230ZM01"."209230CA21".TrfOutResIntlkOk := "TRUE";
END_REGION

REGION Network 33: **** 5.1 - Equations - Interlock **** 230CR22 Transfer IN Set Interlock
   "_209230ZM01"."209230CR22".TrfInSetIntlkOk := "TRUE";
END_REGION

REGION Network 34: **** 5.1 - Equations - Interlock **** 230CR22 Transfer OUT Set Interlock
   "_209230ZM01"."209230CR22".TrfOutSetIntlkOk := "TRUE";
END_REGION

REGION Network 35: **** 5.1 - Equations - Interlock **** 230CR22 Transfer IN Reset Interlock
   "_209230ZM01"."209230CR22".TrfInResIntlkOk := "TRUE";
END_REGION

REGION Network 36: **** 5.1 - Equations - Interlock **** 230CR22 Transfer OUT Reset Interlock
   "_209230ZM01"."209230CR22".TrfOutResIntlkOk := "TRUE";
END_REGION

REGION Network 37: **** 5.2 - Equations - Flow Equation ****230CHB21 Reset (Up) Begin
   "_209230ZM01"."209230CHB21".ResBegin := NOT ("_209230ZS01".AccessStopRequest AND "_209230ZM01"."209230CHB21".SumPosSet) AND "_209230ZM01Orders"."230CHB21Res";
END_REGION

REGION Network 38: **** 5.2 - Equations - Flow Equation **** 230CHB21 Set (Down) Begin
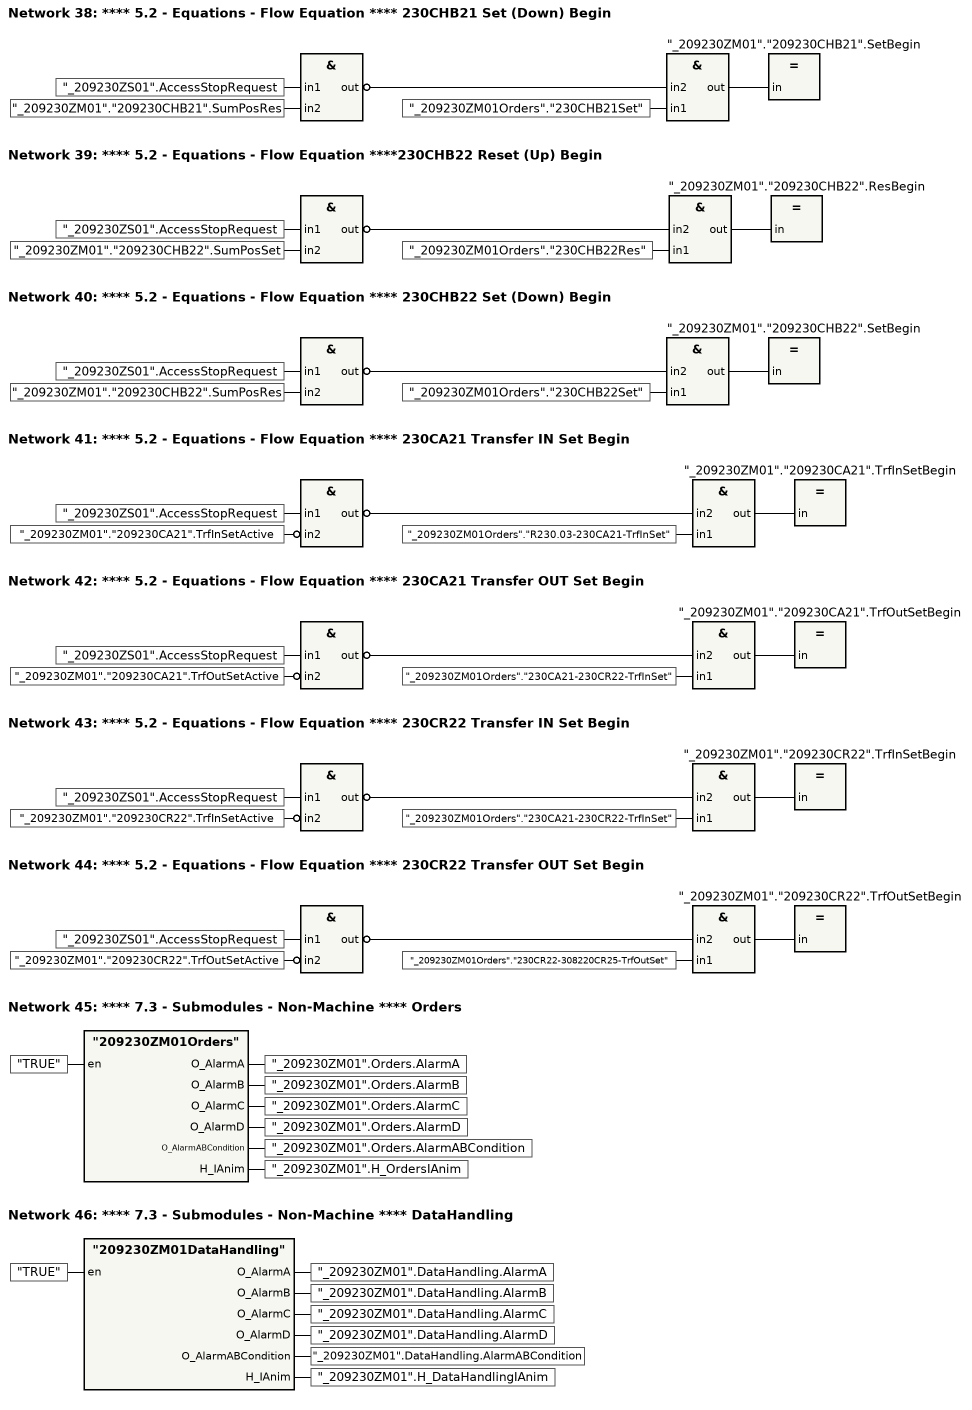
   "_209230ZM01"."209230CHB21".SetBegin := NOT ("_209230ZS01".AccessStopRequest AND "_209230ZM01"."209230CHB21".SumPosRes) AND "_209230ZM01Orders"."230CHB21Set";
END_REGION

REGION Network 39: **** 5.2 - Equations - Flow Equation ****230CHB22 Reset (Up) Begin
   "_209230ZM01"."209230CHB22".ResBegin := NOT ("_209230ZS01".AccessStopRequest AND "_209230ZM01"."209230CHB22".SumPosSet) AND "_209230ZM01Orders"."230CHB22Res";
END_REGION

REGION Network 40: **** 5.2 - Equations - Flow Equation **** 230CHB22 Set (Down) Begin
   "_209230ZM01"."209230CHB22".SetBegin := NOT ("_209230ZS01".AccessStopRequest AND "_209230ZM01"."209230CHB22".SumPosRes) AND "_209230ZM01Orders"."230CHB22Set";
END_REGION

REGION Network 41: **** 5.2 - Equations - Flow Equation **** 230CA21 Transfer IN Set Begin
   "_209230ZM01"."209230CA21".TrfInSetBegin := NOT ("_209230ZS01".AccessStopRequest AND NOT "_209230ZM01"."209230CA21".TrfInSetActive) AND "_209230ZM01Orders"."R230.03-230CA21-TrfInSet";
END_REGION

REGION Network 42: **** 5.2 - Equations - Flow Equation **** 230CA21 Transfer OUT Set Begin
   "_209230ZM01"."209230CA21".TrfOutSetBegin := NOT ("_209230ZS01".AccessStopRequest AND NOT "_209230ZM01"."209230CA21".TrfOutSetActive) AND "_209230ZM01Orders"."230CA21-230CR22-TrfInSet";
END_REGION

REGION Network 43: **** 5.2 - Equations - Flow Equation **** 230CR22 Transfer IN Set Begin
   "_209230ZM01"."209230CR22".TrfInSetBegin := NOT ("_209230ZS01".AccessStopRequest AND NOT "_209230ZM01"."209230CR22".TrfInSetActive) AND "_209230ZM01Orders"."230CA21-230CR22-TrfInSet";
END_REGION

REGION Network 44: **** 5.2 - Equations - Flow Equation **** 230CR22 Transfer OUT Set Begin
   "_209230ZM01"."209230CR22".TrfOutSetBegin := NOT ("_209230ZS01".AccessStopRequest AND NOT "_209230ZM01"."209230CR22".TrfOutSetActive) AND "_209230ZM01Orders"."230CR22-308220CR25-TrfOutSet";
END_REGION

REGION Network 45: **** 7.3 - Submodules - Non-Machine **** Orders
   IF "TRUE" THEN
       "209230ZM01Orders"(O_AlarmA => "_209230ZM01".Orders.AlarmA,
                          O_AlarmB => "_209230ZM01".Orders.AlarmB,
                          O_AlarmC => "_209230ZM01".Orders.AlarmC,
                          O_AlarmD => "_209230ZM01".Orders.AlarmD,
                          O_AlarmABCondition => "_209230ZM01".Orders.AlarmABCondition,
                          H_IAnim => "_209230ZM01".H_OrdersIAnim);
   END_IF;
END_REGION

REGION Network 46: **** 7.3 - Submodules - Non-Machine **** DataHandling
   // Data Handling
   IF "TRUE" THEN
       "209230ZM01DataHandling"(O_AlarmA => "_209230ZM01".DataHandling.AlarmA,
                               O_AlarmB => "_209230ZM01".DataHandling.AlarmB,
                               O_AlarmC => "_209230ZM01".DataHandling.AlarmC,
                               O_AlarmD => "_209230ZM01".DataHandling.AlarmD,
                               O_AlarmABCondition => "_209230ZM01".DataHandling.AlarmABCondition,
                               H_IAnim => "_209230ZM01".H_DataHandlingIAnim);
   END_IF;
END_REGION

REGION Network 47: **** 7.3 - Submodule - Machine **** 230CHB21
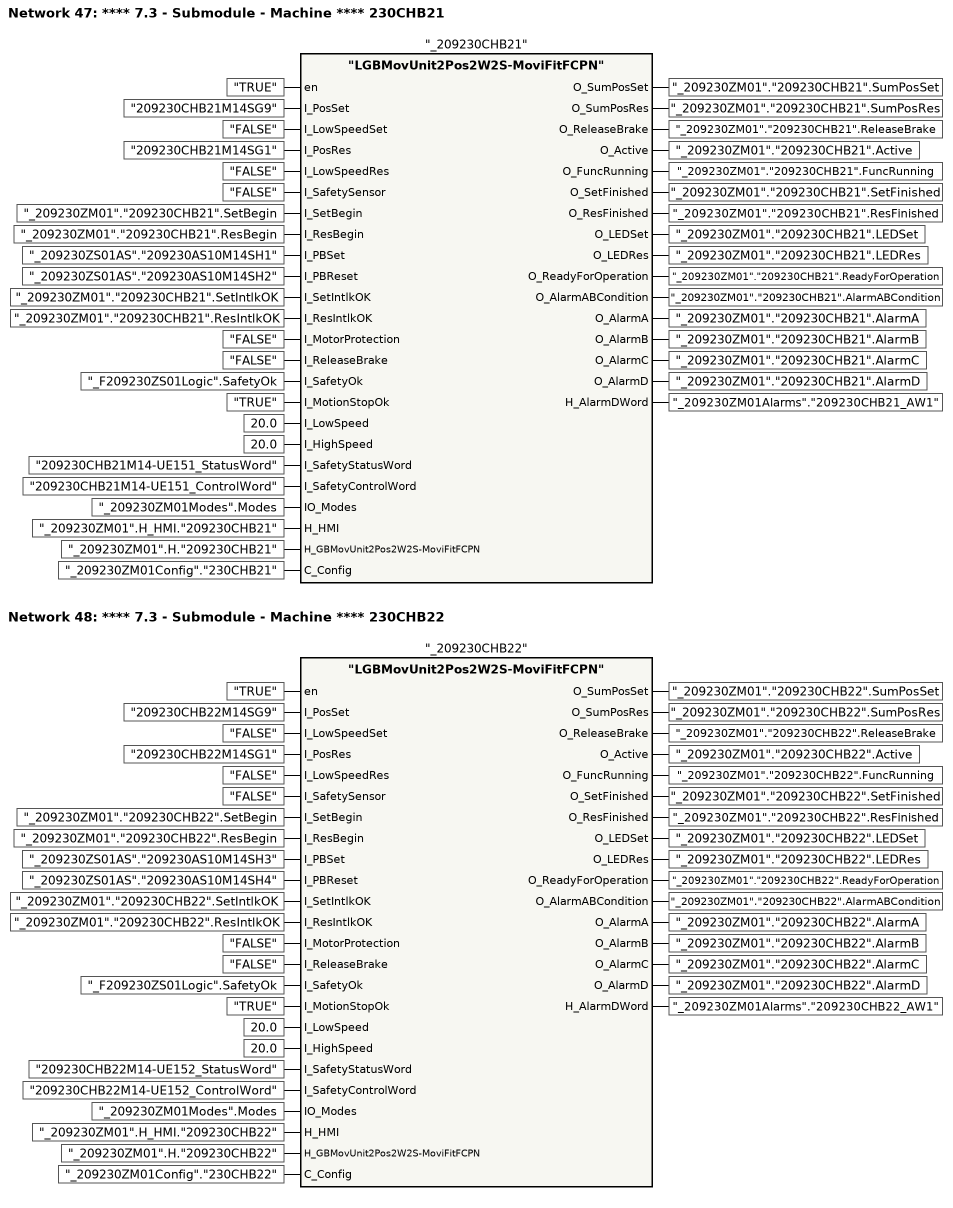
   IF "TRUE" THEN
       "_209230CHB21"(I_PosSet := "209230CHB21M14SG9",   // "LGBMovUnit2Pos2W2S-MoviFitFCPN"
                      I_LowSpeedSet := "FALSE",
                      I_PosRes := "209230CHB21M14SG1",
                      I_LowSpeedRes := "FALSE",
                      I_SafetySensor := "FALSE",
                      I_SetBegin := "_209230ZM01"."209230CHB21".SetBegin,
                      I_ResBegin := "_209230ZM01"."209230CHB21".ResBegin,
                      I_PBSet := "_209230ZS01AS"."209230AS10M14SH1",
                      I_PBReset := "_209230ZS01AS"."209230AS10M14SH2",
                      I_SetIntlkOK := "_209230ZM01"."209230CHB21".SetIntlkOK,
                      I_ResIntlkOK := "_209230ZM01"."209230CHB21".ResIntlkOK,
                      I_MotorProtection := "FALSE",
                      I_ReleaseBrake := "FALSE",
                      I_SafetyOk := "_F209230ZS01Logic".SafetyOk,
                      I_MotionStopOk := "TRUE",
                      I_LowSpeed := 20.0,
                      I_HighSpeed := 20.0,
                      I_SafetyStatusWord := "209230CHB21M14-UE151_StatusWord",
                      I_SafetyControlWord := "209230CHB21M14-UE151_ControlWord",
                      IO_Modes := "_209230ZM01Modes".Modes,
                      H_HMI := "_209230ZM01".H_HMI."209230CHB21",
                      "H_GBMovUnit2Pos2W2S-MoviFitFCPN" := "_209230ZM01".H."209230CHB21",
                      C_Config := "_209230ZM01Config"."230CHB21",
                      O_SumPosSet => "_209230ZM01"."209230CHB21".SumPosSet,
                      O_SumPosRes => "_209230ZM01"."209230CHB21".SumPosRes,
                      O_ReleaseBrake => "_209230ZM01"."209230CHB21".ReleaseBrake,
                      O_Active => "_209230ZM01"."209230CHB21".Active,
                      O_FuncRunning => "_209230ZM01"."209230CHB21".FuncRunning,
                      O_SetFinished => "_209230ZM01"."209230CHB21".SetFinished,
                      O_ResFinished => "_209230ZM01"."209230CHB21".ResFinished,
                      O_LEDSet => "_209230ZM01"."209230CHB21".LEDSet,
                      O_LEDRes => "_209230ZM01"."209230CHB21".LEDRes,
                      O_ReadyForOperation => "_209230ZM01"."209230CHB21".ReadyForOperation,
                      O_AlarmABCondition => "_209230ZM01"."209230CHB21".AlarmABCondition,
                      O_AlarmA => "_209230ZM01"."209230CHB21".AlarmA,
                      O_AlarmB => "_209230ZM01"."209230CHB21".AlarmB,
                      O_AlarmC => "_209230ZM01"."209230CHB21".AlarmC,
                      O_AlarmD => "_209230ZM01"."209230CHB21".AlarmD,
                      H_AlarmDWord => "_209230ZM01Alarms"."209230CHB21_AW1");
   END_IF;
END_REGION

REGION Network 48: **** 7.3 - Submodule - Machine **** 230CHB22
   IF "TRUE" THEN
       "_209230CHB22"(I_PosSet := "209230CHB22M14SG9",   // "LGBMovUnit2Pos2W2S-MoviFitFCPN"
                      I_LowSpeedSet := "FALSE",
                      I_PosRes := "209230CHB22M14SG1",
                      I_LowSpeedRes := "FALSE",
                      I_SafetySensor := "FALSE",
                      I_SetBegin := "_209230ZM01"."209230CHB22".SetBegin,
                      I_ResBegin := "_209230ZM01"."209230CHB22".ResBegin,
                      I_PBSet := "_209230ZS01AS"."209230AS10M14SH3",
                      I_PBReset := "_209230ZS01AS"."209230AS10M14SH4",
                      I_SetIntlkOK := "_209230ZM01"."209230CHB22".SetIntlkOK,
                      I_ResIntlkOK := "_209230ZM01"."209230CHB22".ResIntlkOK,
                      I_MotorProtection := "FALSE",
                      I_ReleaseBrake := "FALSE",
                      I_SafetyOk := "_F209230ZS01Logic".SafetyOk,
                      I_MotionStopOk := "TRUE",
                      I_LowSpeed := 20.0,
                      I_HighSpeed := 20.0,
                      I_SafetyStatusWord := "209230CHB22M14-UE152_StatusWord",
                      I_SafetyControlWord := "209230CHB22M14-UE152_ControlWord",
                      IO_Modes := "_209230ZM01Modes".Modes,
                      H_HMI := "_209230ZM01".H_HMI."209230CHB22",
                      "H_GBMovUnit2Pos2W2S-MoviFitFCPN" := "_209230ZM01".H."209230CHB22",
                      C_Config := "_209230ZM01Config"."230CHB22",
                      O_SumPosSet => "_209230ZM01"."209230CHB22".SumPosSet,
                      O_SumPosRes => "_209230ZM01"."209230CHB22".SumPosRes,
                      O_ReleaseBrake => "_209230ZM01"."209230CHB22".ReleaseBrake,
                      O_Active => "_209230ZM01"."209230CHB22".Active,
                      O_FuncRunning => "_209230ZM01"."209230CHB22".FuncRunning,
                      O_SetFinished => "_209230ZM01"."209230CHB22".SetFinished,
                      O_ResFinished => "_209230ZM01"."209230CHB22".ResFinished,
                      O_LEDSet => "_209230ZM01"."209230CHB22".LEDSet,
                      O_LEDRes => "_209230ZM01"."209230CHB22".LEDRes,
                      O_ReadyForOperation => "_209230ZM01"."209230CHB22".ReadyForOperation,
                      O_AlarmABCondition => "_209230ZM01"."209230CHB22".AlarmABCondition,
                      O_AlarmA => "_209230ZM01"."209230CHB22".AlarmA,
                      O_AlarmB => "_209230ZM01"."209230CHB22".AlarmB,
                      O_AlarmC => "_209230ZM01"."209230CHB22".AlarmC,
                      O_AlarmD => "_209230ZM01"."209230CHB22".AlarmD,
                      H_AlarmDWord => "_209230ZM01Alarms"."209230CHB22_AW1");
   END_IF;
END_REGION

REGION Network 49: **** 7.3 - Submodule - Machine **** 230CA21
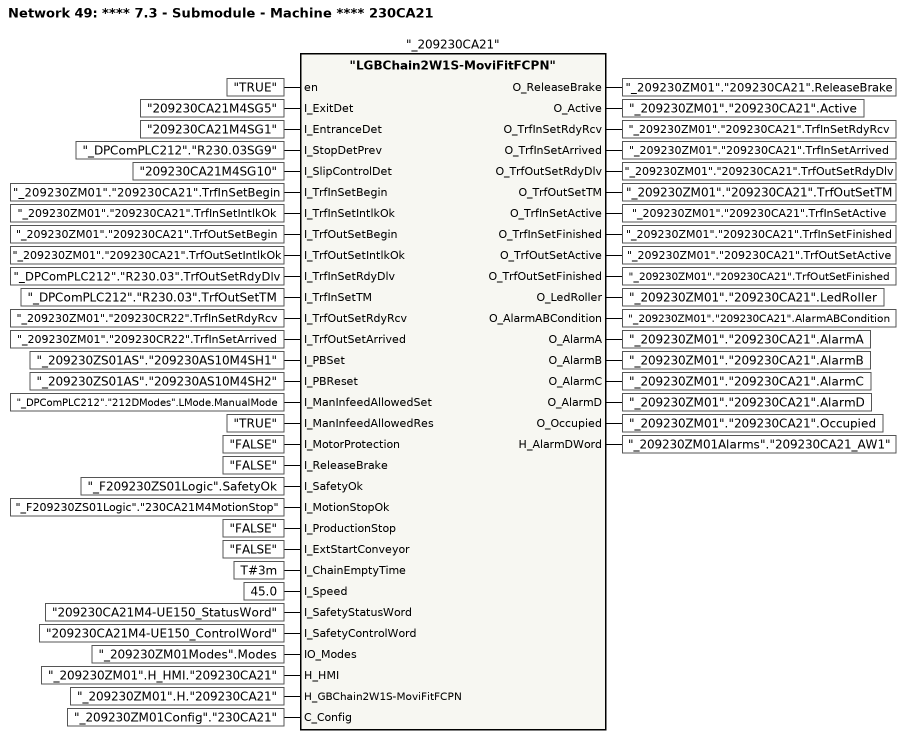
   IF "TRUE" THEN
       "_209230CA21"(I_ExitDet := "209230CA21M4SG5",   // "LGBChain2W1S-MoviFitFCPN"
                     I_EntranceDet := "209230CA21M4SG1",
                     I_StopDetPrev := "_DPComPLC212"."R230.03SG9",
                     I_SlipControlDet := "209230CA21M4SG10",
                     I_TrfInSetBegin := "_209230ZM01"."209230CA21".TrfInSetBegin,
                     I_TrfInSetIntlkOk := "_209230ZM01"."209230CA21".TrfInSetIntlkOk,
                     I_TrfOutSetBegin := "_209230ZM01"."209230CA21".TrfOutSetBegin,
                     I_TrfOutSetIntlkOk := "_209230ZM01"."209230CA21".TrfOutSetIntlkOk,
                     I_TrfInSetRdyDlv := "_DPComPLC212"."R230.03".TrfOutSetRdyDlv,
                     I_TrfInSetTM := "_DPComPLC212"."R230.03".TrfOutSetTM,
                     I_TrfOutSetRdyRcv := "_209230ZM01"."209230CR22".TrfInSetRdyRcv,
                     I_TrfOutSetArrived := "_209230ZM01"."209230CR22".TrfInSetArrived,
                     I_PBSet := "_209230ZS01AS"."209230AS10M4SH1",
                     I_PBReset := "_209230ZS01AS"."209230AS10M4SH2",
                     I_ManInfeedAllowedSet := "_DPComPLC212"."212DModes".LMode.ManualMode,
                     I_ManInfeedAllowedRes := "TRUE",
                     I_MotorProtection := "FALSE",
                     I_ReleaseBrake := "FALSE",
                     I_SafetyOk := "_F209230ZS01Logic".SafetyOk,
                     I_MotionStopOk := "_F209230ZS01Logic"."230CA21M4MotionStop",
                     I_ProductionStop := "FALSE",
                     I_ExtStartConveyor := "FALSE",
                     I_ChainEmptyTime := T#3m,
                     I_Speed := 45.0,
                     I_SafetyStatusWord := "209230CA21M4-UE150_StatusWord",
                     I_SafetyControlWord := "209230CA21M4-UE150_ControlWord",
                     IO_Modes := "_209230ZM01Modes".Modes,
                     H_HMI := "_209230ZM01".H_HMI."209230CA21",
                     "H_GBChain2W1S-MoviFitFCPN" := "_209230ZM01".H."209230CA21",
                     C_Config := "_209230ZM01Config"."230CA21",
                     O_ReleaseBrake => "_209230ZM01"."209230CA21".ReleaseBrake,
                     O_Active => "_209230ZM01"."209230CA21".Active,
                     O_TrfInSetRdyRcv => "_209230ZM01"."209230CA21".TrfInSetRdyRcv,
                     O_TrfInSetArrived => "_209230ZM01"."209230CA21".TrfInSetArrived,
                     O_TrfOutSetRdyDlv => "_209230ZM01"."209230CA21".TrfOutSetRdyDlv,
                     O_TrfOutSetTM => "_209230ZM01"."209230CA21".TrfOutSetTM,
                     O_TrfInSetActive => "_209230ZM01"."209230CA21".TrfInSetActive,
                     O_TrfInSetFinished => "_209230ZM01"."209230CA21".TrfInSetFinished,
                     O_TrfOutSetActive => "_209230ZM01"."209230CA21".TrfOutSetActive,
                     O_TrfOutSetFinished => "_209230ZM01"."209230CA21".TrfOutSetFinished,
                     O_LedRoller => "_209230ZM01"."209230CA21".LedRoller,
                     O_AlarmABCondition => "_209230ZM01"."209230CA21".AlarmABCondition,
                     O_AlarmA => "_209230ZM01"."209230CA21".AlarmA,
                     O_AlarmB => "_209230ZM01"."209230CA21".AlarmB,
                     O_AlarmC => "_209230ZM01"."209230CA21".AlarmC,
                     O_AlarmD => "_209230ZM01"."209230CA21".AlarmD,
                     O_Occupied => "_209230ZM01"."209230CA21".Occupied,
                     H_AlarmDWord => "_209230ZM01Alarms"."209230CA21_AW1");
   END_IF;
END_REGION

REGION Network 50: **** 7.3 - Submodule - Machine **** 230CR22
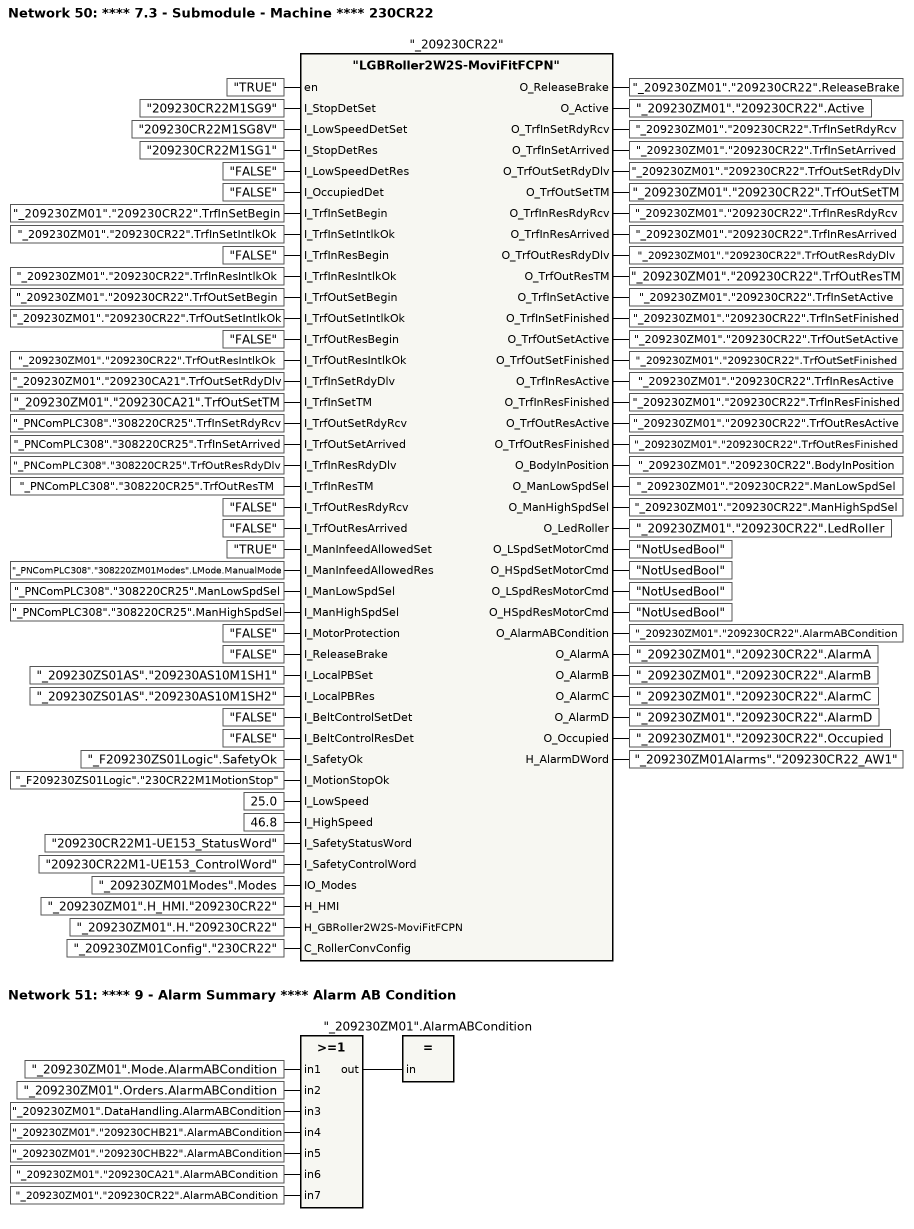
   IF "TRUE" THEN
       "_209230CR22"(I_StopDetSet := "209230CR22M1SG9",   // "LGBRoller2W2S-MoviFitFCPN"
                     I_LowSpeedDetSet := "209230CR22M1SG8V",
                     I_StopDetRes := "209230CR22M1SG1",
                     I_LowSpeedDetRes := "FALSE",
                     I_OccupiedDet := "FALSE",
                     I_TrfInSetBegin := "_209230ZM01"."209230CR22".TrfInSetBegin,
                     I_TrfInSetIntlkOk := "_209230ZM01"."209230CR22".TrfInSetIntlkOk,
                     I_TrfInResBegin := "FALSE",
                     I_TrfInResIntlkOk := "_209230ZM01"."209230CR22".TrfInResIntlkOk,
                     I_TrfOutSetBegin := "_209230ZM01"."209230CR22".TrfOutSetBegin,
                     I_TrfOutSetIntlkOk := "_209230ZM01"."209230CR22".TrfOutSetIntlkOk,
                     I_TrfOutResBegin := "FALSE",
                     I_TrfOutResIntlkOk := "_209230ZM01"."209230CR22".TrfOutResIntlkOk,
                     I_TrfInSetRdyDlv := "_209230ZM01"."209230CA21".TrfOutSetRdyDlv,
                     I_TrfInSetTM := "_209230ZM01"."209230CA21".TrfOutSetTM,
                     I_TrfOutSetRdyRcv := "_PNComPLC308"."308220CR25".TrfInSetRdyRcv,
                     I_TrfOutSetArrived := "_PNComPLC308"."308220CR25".TrfInSetArrived,
                     I_TrfInResRdyDlv := "_PNComPLC308"."308220CR25".TrfOutResRdyDlv,
                     I_TrfInResTM := "_PNComPLC308"."308220CR25".TrfOutResTM,
                     I_TrfOutResRdyRcv := "FALSE",
                     I_TrfOutResArrived := "FALSE",
                     I_ManInfeedAllowedSet := "TRUE",
                     I_ManInfeedAllowedRes := "_PNComPLC308"."308220ZM01Modes".LMode.ManualMode,
                     I_ManLowSpdSel := "_PNComPLC308"."308220CR25".ManLowSpdSel,
                     I_ManHighSpdSel := "_PNComPLC308"."308220CR25".ManHighSpdSel,
                     I_MotorProtection := "FALSE",
                     I_ReleaseBrake := "FALSE",
                     I_LocalPBSet := "_209230ZS01AS"."209230AS10M1SH1",
                     I_LocalPBRes := "_209230ZS01AS"."209230AS10M1SH2",
                     I_BeltControlSetDet := "FALSE",
                     I_BeltControlResDet := "FALSE",
                     I_SafetyOk := "_F209230ZS01Logic".SafetyOk,
                     I_MotionStopOk := "_F209230ZS01Logic"."230CR22M1MotionStop",
                     I_LowSpeed := 25.0,
                     I_HighSpeed := 46.8,
                     I_SafetyStatusWord := "209230CR22M1-UE153_StatusWord",
                     I_SafetyControlWord := "209230CR22M1-UE153_ControlWord",
                     IO_Modes := "_209230ZM01Modes".Modes,
                     H_HMI := "_209230ZM01".H_HMI."209230CR22",
                     "H_GBRoller2W2S-MoviFitFCPN" := "_209230ZM01".H."209230CR22",
                     C_RollerConvConfig := "_209230ZM01Config"."230CR22",
                     O_ReleaseBrake => "_209230ZM01"."209230CR22".ReleaseBrake,
                     O_Active => "_209230ZM01"."209230CR22".Active,
                     O_TrfInSetRdyRcv => "_209230ZM01"."209230CR22".TrfInSetRdyRcv,
                     O_TrfInSetArrived => "_209230ZM01"."209230CR22".TrfInSetArrived,
                     O_TrfOutSetRdyDlv => "_209230ZM01"."209230CR22".TrfOutSetRdyDlv,
                     O_TrfOutSetTM => "_209230ZM01"."209230CR22".TrfOutSetTM,
                     O_TrfInResRdyRcv => "_209230ZM01"."209230CR22".TrfInResRdyRcv,
                     O_TrfInResArrived => "_209230ZM01"."209230CR22".TrfInResArrived,
                     O_TrfOutResRdyDlv => "_209230ZM01"."209230CR22".TrfOutResRdyDlv,
                     O_TrfOutResTM => "_209230ZM01"."209230CR22".TrfOutResTM,
                     O_TrfInSetActive => "_209230ZM01"."209230CR22".TrfInSetActive,
                     O_TrfInSetFinished => "_209230ZM01"."209230CR22".TrfInSetFinished,
                     O_TrfOutSetActive => "_209230ZM01"."209230CR22".TrfOutSetActive,
                     O_TrfOutSetFinished => "_209230ZM01"."209230CR22".TrfOutSetFinished,
                     O_TrfInResActive => "_209230ZM01"."209230CR22".TrfInResActive,
                     O_TrfInResFinished => "_209230ZM01"."209230CR22".TrfInResFinished,
                     O_TrfOutResActive => "_209230ZM01"."209230CR22".TrfOutResActive,
                     O_TrfOutResFinished => "_209230ZM01"."209230CR22".TrfOutResFinished,
                     O_BodyInPosition => "_209230ZM01"."209230CR22".BodyInPosition,
                     O_ManLowSpdSel => "_209230ZM01"."209230CR22".ManLowSpdSel,
                     O_ManHighSpdSel => "_209230ZM01"."209230CR22".ManHighSpdSel,
                     O_LedRoller => "_209230ZM01"."209230CR22".LedRoller,
                     O_LSpdSetMotorCmd => "NotUsedBool",
                     O_HSpdSetMotorCmd => "NotUsedBool",
                     O_LSpdResMotorCmd => "NotUsedBool",
                     O_HSpdResMotorCmd => "NotUsedBool",
                     O_AlarmABCondition => "_209230ZM01"."209230CR22".AlarmABCondition,
                     O_AlarmA => "_209230ZM01"."209230CR22".AlarmA,
                     O_AlarmB => "_209230ZM01"."209230CR22".AlarmB,
                     O_AlarmC => "_209230ZM01"."209230CR22".AlarmC,
                     O_AlarmD => "_209230ZM01"."209230CR22".AlarmD,
                     O_Occupied => "_209230ZM01"."209230CR22".Occupied,
                     H_AlarmDWord => "_209230ZM01Alarms"."209230CR22_AW1");
   END_IF;
END_REGION

REGION Network 51: **** 9 - Alarm Summary **** Alarm AB Condition
   // Alarm AB condition
   "_209230ZM01".AlarmABCondition := "_209230ZM01".Mode.AlarmABCondition OR "_209230ZM01".Orders.AlarmABCondition OR "_209230ZM01".DataHandling.AlarmABCondition OR "_209230ZM01"."209230CHB21".AlarmABCondition OR "_209230ZM01"."209230CHB22".AlarmABCondition OR "_209230ZM01"."209230CA21".AlarmABCondition OR "_209230ZM01"."209230CR22".AlarmABCondition;
END_REGION

REGION Network 52: **** 9 - Alarm Summary **** Alarm A
   // Summary of alarms A
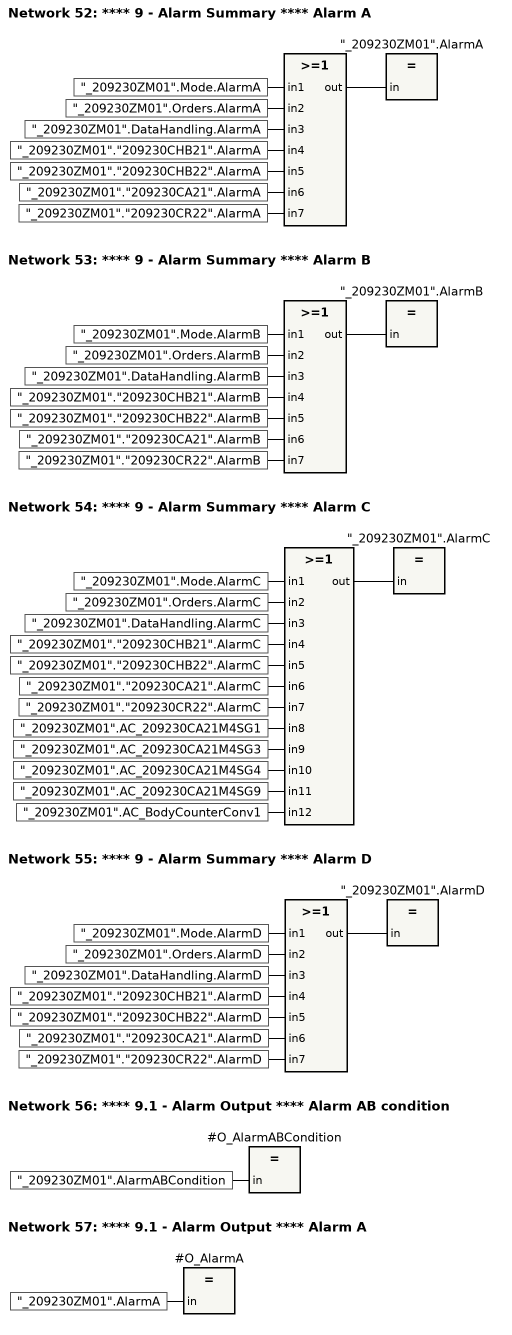
   "_209230ZM01".AlarmA := "_209230ZM01".Mode.AlarmA OR "_209230ZM01".Orders.AlarmA OR "_209230ZM01".DataHandling.AlarmA OR "_209230ZM01"."209230CHB21".AlarmA OR "_209230ZM01"."209230CHB22".AlarmA OR "_209230ZM01"."209230CA21".AlarmA OR "_209230ZM01"."209230CR22".AlarmA;
END_REGION

REGION Network 53: **** 9 - Alarm Summary **** Alarm B
   // Summary of alarms B
   "_209230ZM01".AlarmB := "_209230ZM01".Mode.AlarmB OR "_209230ZM01".Orders.AlarmB OR "_209230ZM01".DataHandling.AlarmB OR "_209230ZM01"."209230CHB21".AlarmB OR "_209230ZM01"."209230CHB22".AlarmB OR "_209230ZM01"."209230CA21".AlarmB OR "_209230ZM01"."209230CR22".AlarmB;
END_REGION

REGION Network 54: **** 9 - Alarm Summary **** Alarm C
   // Summary of alarms C
   "_209230ZM01".AlarmC := "_209230ZM01".Mode.AlarmC OR "_209230ZM01".Orders.AlarmC OR "_209230ZM01".DataHandling.AlarmC OR "_209230ZM01"."209230CHB21".AlarmC OR "_209230ZM01"."209230CHB22".AlarmC OR "_209230ZM01"."209230CA21".AlarmC OR "_209230ZM01"."209230CR22".AlarmC OR "_209230ZM01".AC_209230CA21M4SG1 OR "_209230ZM01".AC_209230CA21M4SG3 OR "_209230ZM01".AC_209230CA21M4SG4 OR "_209230ZM01".AC_209230CA21M4SG9 OR "_209230ZM01".AC_BodyCounterConv1;
END_REGION

REGION Network 55: **** 9 - Alarm Summary **** Alarm D
   // Summary of alarms D
   "_209230ZM01".AlarmD := "_209230ZM01".Mode.AlarmD OR "_209230ZM01".Orders.AlarmD OR "_209230ZM01".DataHandling.AlarmD OR "_209230ZM01"."209230CHB21".AlarmD OR "_209230ZM01"."209230CHB22".AlarmD OR "_209230ZM01"."209230CA21".AlarmD OR "_209230ZM01"."209230CR22".AlarmD;
END_REGION

REGION Network 56: **** 9.1 - Alarm Output **** Alarm AB condition
   // Alarm AB condition
   #O_AlarmABCondition := "_209230ZM01".AlarmABCondition;
END_REGION

REGION Network 57: **** 9.1 - Alarm Output **** Alarm A
   // Output Alarm A
   #O_AlarmA := "_209230ZM01".AlarmA;
END_REGION

REGION Network 58: **** 9.1 - Alarm Output **** Alarm B
   // Output Alarm B
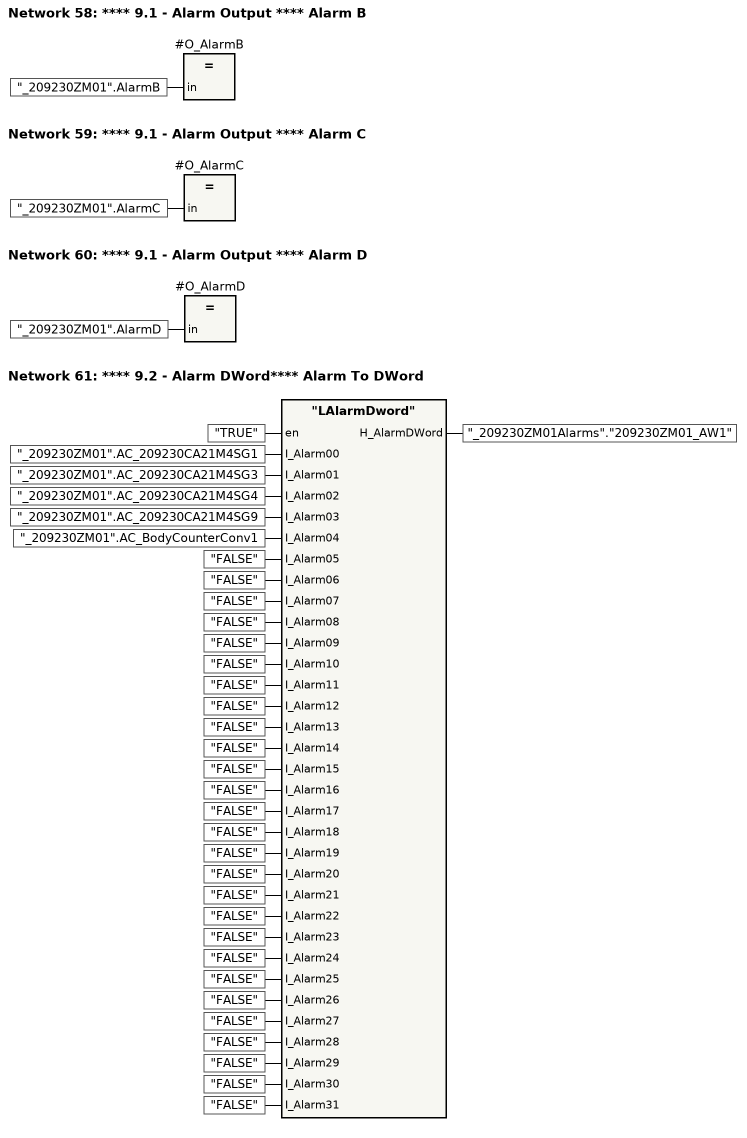
   #O_AlarmB := "_209230ZM01".AlarmB;
END_REGION

REGION Network 59: **** 9.1 - Alarm Output **** Alarm C
   // Output Alarm A
   #O_AlarmC := "_209230ZM01".AlarmC;
END_REGION

REGION Network 60: **** 9.1 - Alarm Output **** Alarm D
   // Output Alarm D
   #O_AlarmD := "_209230ZM01".AlarmD;
END_REGION

REGION Network 61: **** 9.2 - Alarm DWord**** Alarm To DWord
   // Alarm Word
   IF "TRUE" THEN
       "LAlarmDword"(I_Alarm00 := "_209230ZM01".AC_209230CA21M4SG1,
                     I_Alarm01 := "_209230ZM01".AC_209230CA21M4SG3,
                     I_Alarm02 := "_209230ZM01".AC_209230CA21M4SG4,
                     I_Alarm03 := "_209230ZM01".AC_209230CA21M4SG9,
                     I_Alarm04 := "_209230ZM01".AC_BodyCounterConv1,
                     I_Alarm05 := "FALSE",
                     I_Alarm06 := "FALSE",
                     I_Alarm07 := "FALSE",
                     I_Alarm08 := "FALSE",
                     I_Alarm09 := "FALSE",
                     I_Alarm10 := "FALSE",
                     I_Alarm11 := "FALSE",
                     I_Alarm12 := "FALSE",
                     I_Alarm13 := "FALSE",
                     I_Alarm14 := "FALSE",
                     I_Alarm15 := "FALSE",
                     I_Alarm16 := "FALSE",
                     I_Alarm17 := "FALSE",
                     I_Alarm18 := "FALSE",
                     I_Alarm19 := "FALSE",
                     I_Alarm20 := "FALSE",
                     I_Alarm21 := "FALSE",
                     I_Alarm22 := "FALSE",
                     I_Alarm23 := "FALSE",
                     I_Alarm24 := "FALSE",
                     I_Alarm25 := "FALSE",
                     I_Alarm26 := "FALSE",
                     I_Alarm27 := "FALSE",
                     I_Alarm28 := "FALSE",
                     I_Alarm29 := "FALSE",
                     I_Alarm30 := "FALSE",
                     I_Alarm31 := "FALSE",
                     H_AlarmDWord => "_209230ZM01Alarms"."209230ZM01_AW1");
   END_IF;
END_REGION
END_FUNCTION
